# B&R Automation Studio project TD52 (part 57)

#### HiContr.h
```c
/********************************************************************
 * COPYRIGHT -- Bernecker + Rainer Industrie-Elektronik Ges.m.b.H.
 ********************************************************************
 * Program: HiContr
 * File: HiContr.h
 * Author: 106001702
 * Created: Wed Nov 09 12:46:00 2011
 ********************************************************************
 * Header for program HiContr
 ********************************************************************
 * Generated with B&R Automation Studio Target for Simulink V4.2
 * (ERT based)
 ********************************************************************/

#ifndef RTW_HEADER_HiContr_h_
#define RTW_HEADER_HiContr_h_
#ifndef HiContr_COMMON_INCLUDES_
# define HiContr_COMMON_INCLUDES_
#include <math.h>
#include "rtwtypes.h"
#endif                                 /* HiContr_COMMON_INCLUDES_ */

#include "HiContr_types.h"
#include "lHiContr.h"

/* Macros for accessing real-time model data structure */
#ifndef rtmGetErrorStatus
# define rtmGetErrorStatus(rtm)        ((void*) 0)
#endif

#ifndef rtmSetErrorStatus
# define rtmSetErrorStatus(rtm, val)   ((void) 0)
#endif

#ifndef rtmGetStopRequested
# define rtmGetStopRequested(rtm)      ((void*) 0)
#endif

#ifndef MIN
#define MIN(a,b)                       ((a) < (b) ? (a) : (b))
#endif

#ifndef MAX
#define MAX(a,b)                       ((a) > (b) ? (a) : (b))
#endif

/* Block signals (auto storage) */

/* Block states (auto storage) for system '<Root>' */

/* Block signals (auto storage) */
extern BlockIO_HiContr HiContr_B;

/* Block states (auto storage) */
extern D_Work_HiContr HiContr_DWork;

/* Model entry point functions */
extern void HiContr_initialize(struct HiContr* inst);
extern void HiContr_step(struct HiContr* inst);
extern void HiContr_terminate(struct HiContr* inst);

/*-
 * The generated code includes comments that allow you to trace directly
 * back to the appropriate location in the model.  The basic format
 * is <system>/block_name, where system is the system number (uniquely
 * assigned by Simulink) and block_name is the name of the block.
 *
 * Use the MATLAB hilite_system command to trace the generated code back
 * to the model.  For example,
 *
 * hilite_system('<S3>')    - opens system 3
 * hilite_system('<S3>/Kp') - opens and selects block Kp which resides in S3
 *
 * Here is the system hierarchy for this model
 *
 * '<Root>' : 'HiContr'
 * '<S1>'   : 'HiContr/Cyl'
 * '<S2>'   : 'HiContr/Model Info'
 * '<S3>'   : 'HiContr/Cyl/DocBlock'
 * '<S4>'   : 'HiContr/Cyl/GICounter1'
 * '<S5>'   : 'HiContr/Cyl/GlowIgn Integrator'
 * '<S6>'   : 'HiContr/Cyl/Misifire Integrator1'
 * '<S7>'   : 'HiContr/Cyl/Model Info'
 * '<S8>'   : 'HiContr/Cyl/MovingAverage and StdDev'
 * '<S9>'   : 'HiContr/Cyl/Saturation Dynamic1'
 * '<S10>'  : 'HiContr/Cyl/Saturation Dynamic2'
 * '<S11>'  : 'HiContr/Cyl/Saturation Dynamic3'
 * '<S12>'  : 'HiContr/Cyl/Saturation Dynamic4'
 * '<S13>'  : 'HiContr/Cyl/Saturation Dynamic5'
 * '<S14>'  : 'HiContr/Cyl/Threshold'
 * '<S15>'  : 'HiContr/Cyl/Threshold2'
 * '<S16>'  : 'HiContr/Cyl/Threshold3'
 * '<S17>'  : 'HiContr/Cyl/Threshold4'
 * '<S18>'  : 'HiContr/Cyl/Threshold5'
 * '<S19>'  : 'HiContr/Cyl/Threshold6'
 * '<S20>'  : 'HiContr/Cyl/Threshold7'
 * '<S21>'  : 'HiContr/Cyl/Weak Combustion Integrator'
 */
#endif                                 /* RTW_HEADER_HiContr_h_ */
```

#### HiContr_private.h
```c
/********************************************************************
 * COPYRIGHT -- Bernecker + Rainer Industrie-Elektronik Ges.m.b.H.
 ********************************************************************
 * Program: HiContr
 * File: HiContr_private.h
 * Author: 106001702
 * Created: Wed Nov 09 12:46:00 2011
 ********************************************************************
 * Header for program HiContr
 ********************************************************************
 * Generated with B&R Automation Studio Target for Simulink V4.2
 * (ERT based)
 ********************************************************************/

#ifndef RTW_HEADER_HiContr_private_h_
#define RTW_HEADER_HiContr_private_h_
#include "rtwtypes.h"
#include <bur/plctypes.h>
#ifndef __RTWTYPES_H__
#error This file requires rtwtypes.h to be included
#else
#ifdef TMWTYPES_PREVIOUSLY_INCLUDED
#error This file requires rtwtypes.h to be included before tmwtypes.h
#else

/* Check for inclusion of an incorrect version of rtwtypes.h */
#ifndef RTWTYPES_ID_C08S16I32L32N32F1
#error This code was generated with a different "rtwtypes.h" than the file included
#endif                                 /* RTWTYPES_ID_C08S16I32L32N32F1 */
#endif                                 /* TMWTYPES_PREVIOUSLY_INCLUDED */
#endif                                 /* __RTWTYPES_H__ */

#ifndef MIN
#define MIN(a,b)                       ((a) < (b) ? (a) : (b))
#endif

#ifndef MAX
#define MAX(a,b)                       ((a) > (b) ? (a) : (b))
#endif

/* Imported (extern) block parameters */
extern real32_T GIGain;                /* Variable: GIGain
                                        * Referenced by: '<S1>/GIGain (%*100cycles//events)'
                                        */
extern real32_T GIPowGain;             /* Variable: GIPowGain
                                        * Referenced by: '<S1>/GIPowGain (%Pnom*100cycles//events)'
                                        */
extern real32_T MFGain;                /* Variable: MFGain
                                        * Referenced by: '<S1>/MFGain (%*100cycles//events)'
                                        */
extern real32_T MFGainSkipTdown;       /* Variable: MFGainSkipTdown
                                        * Referenced by: '<S1>/MF_Gain_Skip_Tdown'
                                        */
extern real32_T MFThSkipOff;           /* Variable: MFThSkipOff
                                        * Referenced by: '<S1>/Relay1'
                                        */
extern real32_T MFThSkipOn;            /* Variable: MFThSkipOn
                                        * Referenced by: '<S1>/Relay1'
                                        */
extern real32_T PmaxLimReaHys;         /* Variable: PmaxLimReaHys
                                        * Referenced by: '<S1>/Relay'
                                        */
extern real32_T WCGain;                /* Variable: WCGain
                                        * Referenced by: '<S1>/WCGain (bar*100cycles//events)'
                                        */
extern real32_T WCScaling;             /* Variable: WCScaling
                                        * Referenced by: '<S1>/scaling relative to  Pmax at full load (%//bar)'
                                        */

#endif                                 /* RTW_HEADER_HiContr_private_h_ */
```

#### HiContr_types.h
```c
/********************************************************************
 * COPYRIGHT -- Bernecker + Rainer Industrie-Elektronik Ges.m.b.H.
 ********************************************************************
 * Program: HiContr
 * File: HiContr_types.h
 * Author: 106001702
 * Created: Wed Nov 09 12:46:00 2011
 ********************************************************************
 * Header for program HiContr
 ********************************************************************
 * Generated with B&R Automation Studio Target for Simulink V4.2
 * (ERT based)
 ********************************************************************/

#ifndef RTW_HEADER_HiContr_types_h_
#define RTW_HEADER_HiContr_types_h_
#ifndef MIN
#define MIN(a,b)                       ((a) < (b) ? (a) : (b))
#endif

#ifndef MAX
#define MAX(a,b)                       ((a) > (b) ? (a) : (b))
#endif
#endif                                 /* RTW_HEADER_HiContr_types_h_ */
```

#### rtwtypes.h
```c
/********************************************************************
 * COPYRIGHT -- Bernecker + Rainer Industrie-Elektronik Ges.m.b.H.
 ********************************************************************
 * Program: HiContr
 * File: rtwtypes.h
 * Author: 106001702
 * Created: Wed Nov 09 12:46:00 2011
 ********************************************************************
 * Header for program HiContr
 ********************************************************************
 * Generated with B&R Automation Studio Target for Simulink V4.2
 * (ERT based)
 ********************************************************************/

#ifndef __RTWTYPES_H__
#define __RTWTYPES_H__
#ifndef TRUE
# define TRUE                          (1U)
#endif

#ifndef FALSE
# define FALSE                         (0U)
#endif

#ifndef __TMWTYPES__
#define __TMWTYPES__
#include <limits.h>

/*=======================================================================*
 * Target hardware information
 *   Device type: Intel->x86/Pentium
 *   Number of bits:     char:   8    short:   16    int:  32
 *                       long:  32
 *                       native word size:  32
 *   Byte ordering: LittleEndian
 *   Signed integer division rounds to: Zero
 *   Shift right on a signed integer as arithmetic shift: on
 *=======================================================================*/

/*=======================================================================*
 * Fixed width word size data types:                                     *
 *   int8_T, int16_T, int32_T     - signed 8, 16, or 32 bit integers     *
 *   uint8_T, uint16_T, uint32_T  - unsigned 8, 16, or 32 bit integers   *
 *   real32_T, real64_T           - 32 and 64 bit floating point numbers *
 *=======================================================================*/
typedef signed char int8_T;
typedef unsigned char uint8_T;
typedef short int16_T;
typedef unsigned short uint16_T;
typedef int int32_T;
typedef unsigned int uint32_T;
typedef float real32_T;
typedef double real64_T;

/*===========================================================================*
 * Generic type definitions: real_T, time_T, boolean_T, int_T, uint_T,       *
 *                           ulong_T, char_T and byte_T.                     *
 *===========================================================================*/
typedef double real_T;
typedef double time_T;
typedef unsigned char boolean_T;
typedef int int_T;
typedef unsigned int uint_T;
typedef unsigned long ulong_T;
typedef char char_T;
typedef unsigned char uchar_T;
typedef char_T byte_T;

/*=======================================================================*
 * Min and Max:                                                          *
 *   int8_T, int16_T, int32_T     - signed 8, 16, or 32 bit integers     *
 *   uint8_T, uint16_T, uint32_T  - unsigned 8, 16, or 32 bit integers   *
 *=======================================================================*/
#define MAX_int8_T                     ((int8_T)(127))
#define MIN_int8_T                     ((int8_T)(-128))
#define MAX_uint8_T                    ((uint8_T)(255U))
#define MIN_uint8_T                    ((uint8_T)(0U))
#define MAX_int16_T                    ((int16_T)(32767))
#define MIN_int16_T                    ((int16_T)(-32768))
#define MAX_uint16_T                   ((uint16_T)(65535U))
#define MIN_uint16_T                   ((uint16_T)(0U))
#define MAX_int32_T                    ((int32_T)(2147483647))
#define MIN_int32_T                    ((int32_T)(-2147483647-1))
#define MAX_uint32_T                   ((uint32_T)(0xFFFFFFFFU))
#define MIN_uint32_T                   ((uint32_T)(0U))

/* Logical type definitions */
#if (!defined(__cplusplus)) && (!defined(__true_false_are_keywords))
#  ifndef false
#   define false                       (0U)
#  endif

#  ifndef true
#   define true                        (1U)
#  endif
#endif

/*
 * Simulink Coder assumes the code is compiled on a target using a 2's complement representation
 * for signed integer values.
 */
#if ((SCHAR_MIN + 1) != -SCHAR_MAX)
#error "This code must be compiled using a 2's complement representation for signed integer values"
#endif

/* This ID is used to detect inclusion of an incompatible rtwtypes.h */
#define RTWTYPES_ID_C08S16I32L32N32F1
#else                                  /* __TMWTYPES__ */
#define TMWTYPES_PREVIOUSLY_INCLUDED
#endif                                 /* __TMWTYPES__ */

/* Block D-Work pointer type */
typedef void * pointer_T;

/* Simulink specific types */
#ifndef __SIMSTRUC_TYPES_H__
#define __SIMSTRUC_TYPES_H__

/* Trigger directions: falling, either, and rising */
typedef enum {
  FALLING_ZERO_CROSSING = -1,
  ANY_ZERO_CROSSING = 0,
  RISING_ZERO_CROSSING = 1
} ZCDirection;

/* Previous state of a trigger signal */
typedef uint8_T ZCSigState;

/* Initial value of a trigger zero crossing signal */
#define UNINITIALIZED_ZCSIG            0x03U
#define NEG_ZCSIG                      0x02U
#define POS_ZCSIG                      0x01U
#define ZERO_ZCSIG                     0x00U

/* Current state of a trigger signal */
typedef enum {
  FALLING_ZCEVENT = -1,
  NO_ZCEVENT = 0,
  RISING_ZCEVENT = 1
} ZCEventType;

#endif                                 /* __SIMSTRUC_TYPES_H__ */
#endif                                 /* __RTWTYPES_H__ */

#ifndef MIN
#define MIN(a,b)                       ((a) < (b) ? (a) : (b))
#endif

#ifndef MAX
#define MAX(a,b)                       ((a) > (b) ? (a) : (b))
#endif
```

#### HiContr.c
```c
/********************************************************************
 * COPYRIGHT -- Bernecker + Rainer Industrie-Elektronik Ges.m.b.H.
 ********************************************************************
 * Program: HiContr
 * File: HiContr.c
 * Author: 106001702
 * Created: Wed Nov 09 12:46:00 2011
 ********************************************************************
 * Implementation of program HiContr
 ********************************************************************
 * Generated with B&R Automation Studio Target for Simulink V4.2
 * (ERT based)
 ********************************************************************/
#include "HiContr.h"
#include "HiContr_private.h"

/*  Defines */

/*  Data Types */

/**************************** GLOBAL DATA *************************************/
/*  Definitions */

/* Block signals (auto storage) */

/* Block states (auto storage) */

/*  Declarations  */

/***************************** FILE SCOPE DATA ********************************/

/*************************** FUNCTIONS ****************************************/

/* Model step function */
void HiContr_step(struct HiContr* inst)
{
  /* local block i/o variables */
  boolean_T rtb_Compare_j;
  real32_T rtb_Switch1;
  boolean_T rtb_Compare;
  boolean_T rtb_LogicalOperator6;
  real32_T rtb_invert;
  boolean_T rtb_LogicalOperator3;
  real_T rtb_Divide3_g;
  real32_T rtb_MathFunction[100];
  real32_T rtb_Sum;
  real32_T rtb_Divide2;
  real32_T rtb_Add7;
  boolean_T rtb_LogicalOperator1;
  boolean_T rtb_LogicalOperator11;
  boolean_T rtb_LogicalOperator;
  boolean_T rtb_BitwiseOperator2;
  boolean_T rtb_BitwiseOperator1;
  real32_T rtb_Add8;
  real_T rtb_Divide3_d;
  real_T rtb_Divide3_p;
  real_T rtb_Add;
  int32_T i;
  int16_T tmp;

  /* S-Function (bur_in): '<S1>/Input17' */
  inst->bur_HiContr_B.Input17 = inst->GIThPIDUR;

  /* S-Function (bur_in): '<Root>/Input5' */
  inst->bur_HiContr_B.Input5_c = inst->EngStopErrAck;

  /* DiscreteIntegrator: '<S5>/Discrete-Time Integrator' */
  if (inst->bur_HiContr_B.Input5_c || (inst->bur_HiContr_DWork.DiscreteTimeIntegrator_PrevRese != 0))
  {
    inst->bur_HiContr_DWork.DiscreteTimeIntegrator_DSTATE = 0.0F;
  }

  if (inst->bur_HiContr_DWork.DiscreteTimeIntegrator_DSTATE >= 100.0F) {
    inst->bur_HiContr_DWork.DiscreteTimeIntegrator_DSTATE = 100.0F;
  } else {
    if (inst->bur_HiContr_DWork.DiscreteTimeIntegrator_DSTATE <= 0.0F) {
      inst->bur_HiContr_DWork.DiscreteTimeIntegrator_DSTATE = 0.0F;
    }
  }

  inst->bur_HiContr_B.DiscreteTimeIntegrator = inst->bur_HiContr_DWork.DiscreteTimeIntegrator_DSTATE;

  /* End of DiscreteIntegrator: '<S5>/Discrete-Time Integrator' */

  /* Sum: '<S1>/Add5' */
  rtb_Switch1 = inst->bur_HiContr_B.DiscreteTimeIntegrator - inst->bur_HiContr_B.Input17;

  /* S-Function (bur_in): '<Root>/Input9' */
  inst->bur_HiContr_B.Input9_a = inst->GIContrEnable;

  /* Logic: '<S1>/Logical Operator6' incorporates:
   *  Constant: '<S16>/Constant'
   *  RelationalOperator: '<S16>/Compare'
   */
  rtb_LogicalOperator6 = ((rtb_Switch1 > 0.0F) && inst->bur_HiContr_B.Input9_a);

  /* Switch: '<S1>/Switch2' incorporates:
   *  Constant: '<S1>/Constant2'
   */
  if (!rtb_LogicalOperator6) {
    rtb_Switch1 = 0.0F;
  }

  /* End of Switch: '<S1>/Switch2' */

  /* Gain: '<S1>/invert' incorporates:
   *  Gain: '<S1>/GIGain (%*100cycles//events)'
   */
  rtb_invert = -(inst->GIGain * rtb_Switch1);

  /* S-Function (bur_in): '<S1>/Input13' */
  inst->bur_HiContr_B.Input13 = inst->GIPIDURLimMin;

  /* Switch: '<S12>/Switch2' incorporates:
   *  Constant: '<S1>/Constant6'
   *  RelationalOperator: '<S12>/LowerRelop1'
   *  RelationalOperator: '<S12>/UpperRelop'
   *  Switch: '<S12>/Switch'
   */
  if (rtb_invert > 0.0F) {
    inst->bur_HiContr_B.Switch2 = 0.0F;
  } else if (rtb_invert < inst->bur_HiContr_B.Input13) {
    /* Switch: '<S12>/Switch' */
    inst->bur_HiContr_B.Switch2 = inst->bur_HiContr_B.Input13;
  } else {
    inst->bur_HiContr_B.Switch2 = rtb_invert;
  }

  /* End of Switch: '<S12>/Switch2' */

  /* S-Function (bur_out): '<S1>/Output1' */
  inst->PIDUROffsetGI = inst->bur_HiContr_B.Switch2;

  /* S-Function (bur_in): '<S1>/Input11' */
  inst->bur_HiContr_B.Input11 = inst->MFPIDURLimMax;

  /* S-Function (bur_in): '<S1>/Input14' */
  inst->bur_HiContr_B.Input14 = inst->MFThPIDUR;

  /* DiscreteIntegrator: '<S6>/Discrete-Time Integrator' */
  if (inst->bur_HiContr_B.Input5_c || (inst->bur_HiContr_DWork.DiscreteTimeIntegrator_PrevRe_f != 0))
  {
    inst->bur_HiContr_DWork.DiscreteTimeIntegrator_DSTATE_e = 0.0F;
  }

  if (inst->bur_HiContr_DWork.DiscreteTimeIntegrator_DSTATE_e >= 100.0F) {
    inst->bur_HiContr_DWork.DiscreteTimeIntegrator_DSTATE_e = 100.0F;
  } else {
    if (inst->bur_HiContr_DWork.DiscreteTimeIntegrator_DSTATE_e <= 0.0F) {
      inst->bur_HiContr_DWork.DiscreteTimeIntegrator_DSTATE_e = 0.0F;
    }
  }

  inst->bur_HiContr_B.DiscreteTimeIntegrator_d =
    inst->bur_HiContr_DWork.DiscreteTimeIntegrator_DSTATE_e;

  /* End of DiscreteIntegrator: '<S6>/Discrete-Time Integrator' */

  /* Sum: '<S1>/Add2' */
  rtb_Switch1 = inst->bur_HiContr_B.DiscreteTimeIntegrator_d - inst->bur_HiContr_B.Input14;

  /* S-Function (bur_in): '<Root>/Input7' */
  inst->bur_HiContr_B.Input7_c = inst->MFContrEnable;

  /* Logic: '<S1>/Logical Operator3' incorporates:
   *  Constant: '<S14>/Constant'
   *  RelationalOperator: '<S14>/Compare'
   */
  rtb_LogicalOperator3 = ((rtb_Switch1 > 0.0F) && inst->bur_HiContr_B.Input7_c);

  /* Switch: '<S1>/Switch' incorporates:
   *  Constant: '<S1>/Constant'
   */
  if (!rtb_LogicalOperator3) {
    rtb_Switch1 = 0.0F;
  }

  /* End of Switch: '<S1>/Switch' */

  /* Gain: '<S1>/MFGain (%*100cycles//events)' */
  rtb_invert = inst->MFGain * rtb_Switch1;

  /* Switch: '<S9>/Switch2' incorporates:
   *  Constant: '<S1>/Constant7'
   *  RelationalOperator: '<S9>/LowerRelop1'
   *  RelationalOperator: '<S9>/UpperRelop'
   *  Switch: '<S9>/Switch'
   */
  if (rtb_invert > inst->bur_HiContr_B.Input11) {
    inst->bur_HiContr_B.Switch2_e = inst->bur_HiContr_B.Input11;
  } else if (rtb_invert < 0.0F) {
    /* Switch: '<S9>/Switch' incorporates:
     *  Constant: '<S1>/Constant7'
     */
    inst->bur_HiContr_B.Switch2_e = 0.0F;
  } else {
    inst->bur_HiContr_B.Switch2_e = rtb_invert;
  }

  /* End of Switch: '<S9>/Switch2' */

  /* S-Function (bur_out): '<S1>/Output2' */
  inst->PIDUROffsetMF = inst->bur_HiContr_B.Switch2_e;

  /* S-Function (bur_out): '<S1>/Output3' */
  inst->MFIntOut = inst->bur_HiContr_B.DiscreteTimeIntegrator_d;

  /* DiscreteIntegrator: '<S21>/Discrete-Time Integrator' */
  if (inst->bur_HiContr_B.Input5_c || (inst->bur_HiContr_DWork.DiscreteTimeIntegrator_PrevRe_c != 0))
  {
    inst->bur_HiContr_DWork.DiscreteTimeIntegrator_DSTATE_c = 0.0F;
  }

  if (inst->bur_HiContr_DWork.DiscreteTimeIntegrator_DSTATE_c >= 100.0F) {
    inst->bur_HiContr_DWork.DiscreteTimeIntegrator_DSTATE_c = 100.0F;
  } else {
    if (inst->bur_HiContr_DWork.DiscreteTimeIntegrator_DSTATE_c <= 0.0F) {
      inst->bur_HiContr_DWork.DiscreteTimeIntegrator_DSTATE_c = 0.0F;
    }
  }

  inst->bur_HiContr_B.DiscreteTimeIntegrator_l =
    inst->bur_HiContr_DWork.DiscreteTimeIntegrator_DSTATE_c;

  /* End of DiscreteIntegrator: '<S21>/Discrete-Time Integrator' */

  /* S-Function (bur_out): '<S1>/Output4' */
  inst->WCIntOut = inst->bur_HiContr_B.DiscreteTimeIntegrator_l;

  /* S-Function (bur_out): '<S1>/Output5' */
  inst->GIIntOut = inst->bur_HiContr_B.DiscreteTimeIntegrator;

  /* S-Function (bur_in): '<Root>/Input10' */
  inst->bur_HiContr_B.Input10_h = inst->PmaxLimContrEnable;

  /* S-Function (bur_in): '<Root>/Input11' */
  inst->bur_HiContr_B.Input11_h = inst->PmaxLimDiane;

  /* S-Function (bur_in): '<S1>/Input7' */
  inst->bur_HiContr_B.Input7 = inst->PmaxSDLimMar;

  /* Sum: '<S1>/Subtract' */
  rtb_invert = inst->bur_HiContr_B.Input11_h - inst->bur_HiContr_B.Input7;

  /* Sum: '<S8>/Sum of Elements' incorporates:
   *  S-Function (sfix_udelay): '<S8>/Tapped Delay set as N_cyc!!!'
   */
  rtb_Divide3_g = inst->bur_HiContr_DWork.TappedDelaysetasN_cyc_X[0];
  for (i = 0; i < 99; i++) {
    rtb_Divide3_g += (real_T)inst->bur_HiContr_DWork.TappedDelaysetasN_cyc_X[i + 1];
  }

  /* End of Sum: '<S8>/Sum of Elements' */

  /* Product: '<S8>/Divide' incorporates:
   *  Constant: '<S8>/set as Ncyc!!!'
   */
  inst->bur_HiContr_B.Divide = (real32_T)(rtb_Divide3_g / 100.0);

  /* Math: '<S8>/Math Function'
   *
   * About '<S8>/Math Function':
   *  Operator: magnitude^2
   */
  for (i = 0; i < 100; i++) {
    /* Sum: '<S8>/Add' incorporates:
     *  S-Function (sfix_udelay): '<S8>/Tapped Delay set as N_cyc!!!'
     */
    rtb_Switch1 = inst->bur_HiContr_DWork.TappedDelaysetasN_cyc_X[i] - inst->bur_HiContr_B.Divide;
    rtb_MathFunction[i] = rtb_Switch1 * rtb_Switch1;
  }

  /* End of Math: '<S8>/Math Function' */

  /* Sum: '<S8>/Sum of Elements2' */
  rtb_Switch1 = rtb_MathFunction[0];
  for (i = 0; i < 99; i++) {
    rtb_Switch1 += rtb_MathFunction[i + 1];
  }

  /* End of Sum: '<S8>/Sum of Elements2' */

  /* Sqrt: '<S8>/Sqrt' incorporates:
   *  Constant: '<S8>/set as Ncyc!!!'
   *  Product: '<S8>/Divide1'
   */
  inst->bur_HiContr_B.Sqrt = (real32_T)sqrt((real32_T)((real_T)rtb_Switch1 / 100.0));

  /* S-Function (bur_in): '<S1>/Input8' */
  inst->bur_HiContr_B.Input8 = inst->PmaxStdevFact;

  /* Sum: '<S1>/Sum' incorporates:
   *  Product: '<S1>/Product2'
   *  Sum: '<S1>/Add'
   */
  rtb_Sum = rtb_invert - (inst->bur_HiContr_B.Sqrt * inst->bur_HiContr_B.Input8 + inst->bur_HiContr_B.Divide);

  /* S-Function (bur_in): '<S1>/Input9' */
  inst->bur_HiContr_B.Input9 = inst->PmaxContrGain;

  /* Product: '<S1>/Product1' incorporates:
   *  Product: '<S1>/Product3'
   */
  rtb_invert = inst->bur_HiContr_B.Input10_h ? rtb_Sum * inst->bur_HiContr_B.Input9 : 0.0F;

  /* S-Function (bur_in): '<S1>/Input10' */
  inst->bur_HiContr_B.Input10 = inst->PmaxContrLimMin;

  /* Switch: '<S10>/Switch2' incorporates:
   *  Constant: '<S1>/Constant4'
   *  RelationalOperator: '<S10>/LowerRelop1'
   *  RelationalOperator: '<S10>/UpperRelop'
   *  Switch: '<S10>/Switch'
   */
  if (rtb_invert > 0.0F) {
    inst->bur_HiContr_B.Switch2_k = 0.0F;
  } else if (rtb_invert < inst->bur_HiContr_B.Input10) {
    /* Switch: '<S10>/Switch' */
    inst->bur_HiContr_B.Switch2_k = inst->bur_HiContr_B.Input10;
  } else {
    inst->bur_HiContr_B.Switch2_k = rtb_invert;
  }

  /* End of Switch: '<S10>/Switch2' */

  /* S-Function (bur_out): '<S1>/Output6' */
  inst->PIDUROffsetPmax = inst->bur_HiContr_B.Switch2_k;

  /* S-Function (bur_in): '<S1>/Input19' */
  inst->bur_HiContr_B.Input19 = inst->GIThSkipReset;

  /* RelationalOperator: '<S18>/Compare' incorporates:
   *  Constant: '<S18>/Constant'
   *  Sum: '<S1>/Add1'
   */
  rtb_Compare_j = (inst->bur_HiContr_B.DiscreteTimeIntegrator - inst->bur_HiContr_B.Input19 < 0.0F);

  /* DiscreteIntegrator: '<S4>/Discrete-Time Integrator' */
  if (rtb_Compare_j || (inst->bur_HiContr_DWork.DiscreteTimeIntegrator_PrevRe_n != 0)) {
    inst->bur_HiContr_DWork.DiscreteTimeIntegrator_DSTATE_n = 0.0F;
  }

  if (inst->bur_HiContr_DWork.DiscreteTimeIntegrator_DSTATE_n >= 100.0F) {
    inst->bur_HiContr_DWork.DiscreteTimeIntegrator_DSTATE_n = 100.0F;
  } else {
    if (inst->bur_HiContr_DWork.DiscreteTimeIntegrator_DSTATE_n <= 0.0F) {
      inst->bur_HiContr_DWork.DiscreteTimeIntegrator_DSTATE_n = 0.0F;
    }
  }

  inst->bur_HiContr_B.DiscreteTimeIntegrator_dl =
    inst->bur_HiContr_DWork.DiscreteTimeIntegrator_DSTATE_n;

  /* End of DiscreteIntegrator: '<S4>/Discrete-Time Integrator' */

  /* S-Function (bur_out): '<S1>/Output7' */
  inst->GICountOut = inst->bur_HiContr_B.DiscreteTimeIntegrator_dl;

  /* S-Function (bur_out): '<S1>/Output8' */
  inst->PmaxAv = inst->bur_HiContr_B.Divide;

  /* S-Function (bur_out): '<S1>/Output9' */
  inst->PmaxStd = inst->bur_HiContr_B.Sqrt;

  /* S-Function (bur_in): '<S1>/Input16' */
  inst->bur_HiContr_B.Input16 = inst->WCThPmax;

  /* Sum: '<S1>/Add4' */
  rtb_Switch1 = inst->bur_HiContr_B.DiscreteTimeIntegrator_l - inst->bur_HiContr_B.Input16;

  /* S-Function (bur_in): '<S1>/Input18' */
  inst->bur_HiContr_B.Input18 = inst->GIThSkip;

  /* Sum: '<S1>/Add6' */
  rtb_invert = inst->bur_HiContr_B.DiscreteTimeIntegrator - inst->bur_HiContr_B.Input18;

  /* S-Function (bur_in): '<S1>/Input21' */
  inst->bur_HiContr_B.Input21 = inst->GIThCount;

  /* Sum: '<S1>/Add7' */
  rtb_Add7 = inst->bur_HiContr_B.DiscreteTimeIntegrator_dl - inst->bur_HiContr_B.Input21;

  /* Relay: '<S1>/Relay1' */
  if (inst->bur_HiContr_B.DiscreteTimeIntegrator_d >= inst->MFThSkipOn) {
    inst->bur_HiContr_DWork.Relay1_Mode = TRUE;
  } else {
    if (inst->bur_HiContr_B.DiscreteTimeIntegrator_d <= inst->MFThSkipOff) {
      inst->bur_HiContr_DWork.Relay1_Mode = FALSE;
    }
  }

  if (inst->bur_HiContr_DWork.Relay1_Mode) {
    rtb_Divide2 = 1.0F;
  } else {
    rtb_Divide2 = 0.0F;
  }

  /* End of Relay: '<S1>/Relay1' */

  /* Sum: '<S1>/Add8' incorporates:
   *  Constant: '<S1>/Constant3'
   *  Gain: '<S1>/MF_Gain_Skip_Tdown'
   */
  rtb_Add8 = inst->MFGainSkipTdown * rtb_Divide2 + 1.0F;

  /* S-Function (bur_in): '<Root>/Input1' */
  inst->bur_HiContr_B.Input1_h = inst->Misfire2;

  /* S-Function (sfix_bitop): '<S1>/Bitwise Operator' */
  rtb_Compare = !inst->bur_HiContr_B.Input1_h;

  /* S-Function (bur_in): '<Root>/Input20' */
  inst->bur_HiContr_B.Input20_o = inst->Misfire1;

  /* S-Function (sfix_bitop): '<S1>/Bitwise Operator1' */
  rtb_BitwiseOperator1 = !inst->bur_HiContr_B.Input20_o;

  /* RelationalOperator: '<S19>/Compare' incorporates:
   *  Constant: '<S19>/Constant'
   */
  rtb_LogicalOperator1 = (rtb_Add7 > 0.0F);

  /* S-Function (sfix_bitop): '<S1>/Bitwise Operator2' */
  rtb_BitwiseOperator2 = !rtb_LogicalOperator1;

  /* S-Function (bur_in): '<Root>/Input4' */
  inst->bur_HiContr_B.Input4_d = inst->SensSignFault;

  /* S-Function (sfix_bitop): '<S1>/Bitwise Operator3' */
  rtb_LogicalOperator = !inst->bur_HiContr_B.Input4_d;

  /* S-Function (bur_in): '<S1>/Input6' */
  inst->bur_HiContr_B.Input6 = inst->TGICount;

  /* Logic: '<S1>/Logical Operator9' incorporates:
   *  Constant: '<S17>/Constant'
   *  RelationalOperator: '<S17>/Compare'
   */
  rtb_LogicalOperator11 = (inst->bur_HiContr_B.Input9_a && (rtb_invert > 0.0F));

  /* Sum: '<S4>/Add' incorporates:
   *  Constant: '<S1>/Constant9'
   *  Product: '<S4>/Divide'
   *  Product: '<S4>/Divide2'
   */
  rtb_Add = rtb_LogicalOperator11 ? 1.0 / (real_T)inst->bur_HiContr_B.Input6 : 0.0;

  /* Switch: '<S1>/Switch3' incorporates:
   *  Constant: '<S1>/Constant12'
   *  Logic: '<S1>/Logical Operator10'
   */
  if (rtb_LogicalOperator1 && inst->bur_HiContr_B.Input9_a) {
    /* Switch: '<S13>/Switch2' incorporates:
     *  Constant: '<S1>/Constant10'
     *  Constant: '<S1>/Constant11'
     *  RelationalOperator: '<S13>/LowerRelop1'
     *  RelationalOperator: '<S13>/UpperRelop'
     *  Switch: '<S13>/Switch'
     */
    if (rtb_invert > 100.0F) {
      rtb_invert = 100.0F;
    } else {
      if (rtb_invert < 0.0F) {
        /* Switch: '<S13>/Switch' incorporates:
         *  Constant: '<S1>/Constant10'
         */
        rtb_invert = 0.0F;
      }
    }

    /* End of Switch: '<S13>/Switch2' */
  } else {
    rtb_invert = 0.0F;
  }

  /* End of Switch: '<S1>/Switch3' */

  /* Gain: '<S1>/GIPowGain (%Pnom*100cycles//events)' */
  inst->bur_HiContr_B.GIPowGainPnom100cyclesevents = inst->GIPowGain * rtb_invert;

  /* S-Function (bur_in): '<S1>/Input5' */
  inst->bur_HiContr_B.Input5 = inst->TdownGI;

  /* Product: '<S5>/Divide1' incorporates:
   *  Constant: '<S5>/Constant'
   */
  rtb_Divide3_g = 1.0 / (real_T)inst->bur_HiContr_B.Input5;

  /* S-Function (bur_in): '<Root>/Input2' */
  inst->bur_HiContr_B.Input2_g = inst->GlowIgn;

  /* S-Function (bur_in): '<S1>/Input4' */
  inst->bur_HiContr_B.Input4 = inst->TupGI;

  /* Sum: '<S5>/Add' incorporates:
   *  Product: '<S5>/Divide'
   *  Product: '<S5>/Divide2'
   *  Product: '<S5>/Divide3'
   */
  rtb_Divide3_g = (real_T)(rtb_LogicalOperator ? (real32_T)inst->bur_HiContr_B.Input2_g /
    inst->bur_HiContr_B.Input4 : 0.0F) - (rtb_LogicalOperator ? rtb_Divide3_g : 0.0);

  /* S-Function (bur_in): '<S1>/Input1' */
  inst->bur_HiContr_B.Input1 = inst->TdownMF;

  /* S-Function (bur_in): '<S1>/Input12' */
  inst->bur_HiContr_B.Input12 = inst->WCPmaxLimMax;

  /* S-Function (bur_in): '<S1>/Input2' */
  inst->bur_HiContr_B.Input2 = inst->TupWC;

  /* S-Function (bur_in): '<S1>/Input20' */
  inst->bur_HiContr_B.Input20 = inst->TupMF;

  /* S-Function (bur_in): '<S1>/Input3' */
  inst->bur_HiContr_B.Input3 = inst->TdownWC;

  /* Logic: '<S1>/Logical Operator' */
  rtb_LogicalOperator = (inst->bur_HiContr_B.Input20_o && inst->bur_HiContr_B.Input1_h);

  /* Logic: '<S1>/Logical Operator1' */
  rtb_LogicalOperator1 = (inst->bur_HiContr_B.Input20_o && rtb_Compare);

  /* S-Function (bur_in): '<Root>/Input6' */
  inst->bur_HiContr_B.Input6_a = inst->KnockCountMeasAct;

  /* Relay: '<S1>/Relay' */
  if (rtb_Sum >= inst->PmaxLimReaHys) {
    inst->bur_HiContr_DWork.Relay_Mode = TRUE;
  } else {
    if (rtb_Sum <= 0.0F) {
      inst->bur_HiContr_DWork.Relay_Mode = FALSE;
    }
  }

  if (inst->bur_HiContr_DWork.Relay_Mode) {
    tmp = 0;
  } else {
    tmp = 1;
  }

  /* End of Relay: '<S1>/Relay' */

  /* RelationalOperator: '<S20>/Compare' incorporates:
   *  Constant: '<S20>/Constant'
   */
  inst->bur_HiContr_B.Compare = (tmp > 0);

  /* Logic: '<S1>/Logical Operator13' incorporates:
   *  Logic: '<S1>/Logical Operator14'
   *  Logic: '<S1>/Logical Operator5'
   */
  inst->bur_HiContr_B.LogicalOperator13 = ((inst->bur_HiContr_B.Input7_c && (rtb_Divide2 != 0.0F)) ||
                                 (rtb_LogicalOperator11 && rtb_BitwiseOperator2));

  /* S-Function (bur_in): '<Root>/Input12' */
  inst->bur_HiContr_B.Input12_e = inst->SkipCylExt;

  /* Logic: '<S1>/Logical Operator11' incorporates:
   *  Logic: '<S1>/Logical Operator12'
   */
  rtb_LogicalOperator11 = !(inst->bur_HiContr_B.Input6_a || rtb_LogicalOperator6 ||
    inst->bur_HiContr_B.Compare || inst->bur_HiContr_B.Input4_d || (inst->bur_HiContr_B.LogicalOperator13 ||
    inst->bur_HiContr_B.Input12_e));

  /* Logic: '<S1>/Logical Operator2' */
  inst->bur_HiContr_B.LogicalOperator2 = (rtb_BitwiseOperator1 && inst->bur_HiContr_B.Input1_h);

  /* S-Function (bur_in): '<Root>/Input8' */
  inst->bur_HiContr_B.Input8_f = inst->WCContrEnable;

  /* Logic: '<S1>/Logical Operator7' */
  inst->bur_HiContr_B.LogicalOperator7 = (rtb_LogicalOperator3 || rtb_LogicalOperator6 ||
    inst->bur_HiContr_B.Compare || inst->bur_HiContr_B.Input4_d);

  /* Logic: '<S1>/Logical Operator8' */
  inst->bur_HiContr_B.LogicalOperator8 = (rtb_LogicalOperator3 || rtb_LogicalOperator6 ||
    inst->bur_HiContr_B.Compare || inst->bur_HiContr_B.Input4_d);

  /* MinMax: '<S1>/MinMax' */
  if (inst->bur_HiContr_B.Switch2_k <= inst->bur_HiContr_B.Switch2) {
    rtb_Add7 = inst->bur_HiContr_B.Switch2_k;
  } else {
    rtb_Add7 = inst->bur_HiContr_B.Switch2;
  }

  /* Product: '<S6>/Divide3' incorporates:
   *  Constant: '<S6>/Constant'
   *  Product: '<S1>/Product'
   *  Product: '<S6>/Divide1'
   */
  rtb_Divide3_d = 1.0 / (real_T)(inst->bur_HiContr_B.Input1 * rtb_Add8);

  /* Product: '<S6>/Divide2' incorporates:
   *  Product: '<S6>/Divide'
   */
  rtb_Divide2 = rtb_LogicalOperator11 ? (real32_T)rtb_LogicalOperator /
    inst->bur_HiContr_B.Input20 : 0.0F;

  /* Switch: '<S1>/Switch1' incorporates:
   *  Constant: '<S15>/Constant'
   *  Constant: '<S1>/Constant1'
   *  Logic: '<S1>/Logical Operator4'
   *  RelationalOperator: '<S15>/Compare'
   */
  if (!((rtb_Switch1 > 0.0F) && inst->bur_HiContr_B.Input8_f)) {
    rtb_Switch1 = 0.0F;
  }

  /* End of Switch: '<S1>/Switch1' */

  /* Gain: '<S1>/scaling relative to  Pmax at full load (%//bar)' incorporates:
   *  Gain: '<S1>/WCGain (bar*100cycles//events)'
   */
  rtb_invert = inst->WCGain * rtb_Switch1 * inst->WCScaling;

  /* Switch: '<S11>/Switch2' incorporates:
   *  Constant: '<S1>/Constant8'
   *  RelationalOperator: '<S11>/LowerRelop1'
   *  RelationalOperator: '<S11>/UpperRelop'
   *  Switch: '<S11>/Switch'
   */
  if (rtb_invert > inst->bur_HiContr_B.Input12) {
    inst->bur_HiContr_B.Switch2_a = inst->bur_HiContr_B.Input12;
  } else if (rtb_invert < 0.0F) {
    /* Switch: '<S11>/Switch' incorporates:
     *  Constant: '<S1>/Constant8'
     */
    inst->bur_HiContr_B.Switch2_a = 0.0F;
  } else {
    inst->bur_HiContr_B.Switch2_a = rtb_invert;
  }

  /* End of Switch: '<S11>/Switch2' */

  /* Switch: '<S1>/Switch4' incorporates:
   *  MinMax: '<S1>/MinMax'
   */
  if (rtb_Add7 >= 0.0F) {
    inst->bur_HiContr_B.Switch4 = inst->bur_HiContr_B.Switch2_e;
  } else {
    inst->bur_HiContr_B.Switch4 = rtb_Add7;
  }

  /* End of Switch: '<S1>/Switch4' */

  /* Product: '<S21>/Divide3' incorporates:
   *  Constant: '<S21>/Constant'
   *  Product: '<S21>/Divide1'
   */
  rtb_Divide3_p = 1.0 / (real_T)inst->bur_HiContr_B.Input3;

  /* Product: '<S21>/Divide2' incorporates:
   *  Product: '<S21>/Divide'
   */
  rtb_invert = rtb_LogicalOperator11 ? (real32_T)rtb_LogicalOperator1 /
    inst->bur_HiContr_B.Input2 : 0.0F;

  /* S-Function (bur_out): '<Root>/Output1' */
  inst->FaultMFSign = inst->bur_HiContr_B.LogicalOperator2;

  /* S-Function (bur_out): '<Root>/Output2' */
  inst->MFB50Freeze = inst->bur_HiContr_B.LogicalOperator7;

  /* S-Function (bur_out): '<Root>/Output3' */
  inst->OptPIDFreeze = inst->bur_HiContr_B.LogicalOperator8;

  /* S-Function (bur_out): '<Root>/Output4' */
  inst->PIDUROffsetCyl = inst->bur_HiContr_B.Switch4;

  /* S-Function (bur_out): '<Root>/Output6' */
  inst->PmaxStabLayOffset = inst->bur_HiContr_B.Switch2_a;

  /* S-Function (bur_out): '<Root>/Output7' */
  inst->PmaxLimReached = inst->bur_HiContr_B.Compare;

  /* S-Function (bur_out): '<Root>/Output8' */
  inst->SkipCyl = inst->bur_HiContr_B.LogicalOperator13;

  /* S-Function (bur_out): '<Root>/Output9' */
  inst->PowRedCyl = inst->bur_HiContr_B.GIPowGainPnom100cyclesevents;

  /* S-Function (bur_in): '<Root>/Input3' */
  inst->bur_HiContr_B.Input3_g = inst->Pmax;

  /* Update for DiscreteIntegrator: '<S5>/Discrete-Time Integrator' */
  if (!inst->bur_HiContr_B.Input5_c) {
    inst->bur_HiContr_DWork.DiscreteTimeIntegrator_DSTATE += (real32_T)(0.01 *
      rtb_Divide3_g);
    if (inst->bur_HiContr_DWork.DiscreteTimeIntegrator_DSTATE >= 100.0F) {
      inst->bur_HiContr_DWork.DiscreteTimeIntegrator_DSTATE = 100.0F;
    } else {
      if (inst->bur_HiContr_DWork.DiscreteTimeIntegrator_DSTATE <= 0.0F) {
        inst->bur_HiContr_DWork.DiscreteTimeIntegrator_DSTATE = 0.0F;
      }
    }
  }

  if (inst->bur_HiContr_B.Input5_c) {
    inst->bur_HiContr_DWork.DiscreteTimeIntegrator_PrevRese = 1;
  } else {
    inst->bur_HiContr_DWork.DiscreteTimeIntegrator_PrevRese = 0;
  }

  /* End of Update for DiscreteIntegrator: '<S5>/Discrete-Time Integrator' */

  /* Update for DiscreteIntegrator: '<S6>/Discrete-Time Integrator' incorporates:
   *  Sum: '<S6>/Add'
   */
  if (!inst->bur_HiContr_B.Input5_c) {
    inst->bur_HiContr_DWork.DiscreteTimeIntegrator_DSTATE_e += (real32_T)(((real_T)
      rtb_Divide2 - rtb_Divide3_d) * 0.01);
    if (inst->bur_HiContr_DWork.DiscreteTimeIntegrator_DSTATE_e >= 100.0F) {
      inst->bur_HiContr_DWork.DiscreteTimeIntegrator_DSTATE_e = 100.0F;
    } else {
      if (inst->bur_HiContr_DWork.DiscreteTimeIntegrator_DSTATE_e <= 0.0F) {
        inst->bur_HiContr_DWork.DiscreteTimeIntegrator_DSTATE_e = 0.0F;
      }
    }
  }

  if (inst->bur_HiContr_B.Input5_c) {
    inst->bur_HiContr_DWork.DiscreteTimeIntegrator_PrevRe_f = 1;
  } else {
    inst->bur_HiContr_DWork.DiscreteTimeIntegrator_PrevRe_f = 0;
  }

  /* End of Update for DiscreteIntegrator: '<S6>/Discrete-Time Integrator' */

  /* Update for DiscreteIntegrator: '<S21>/Discrete-Time Integrator' incorporates:
   *  Sum: '<S21>/Add'
   */
  if (!inst->bur_HiContr_B.Input5_c) {
    inst->bur_HiContr_DWork.DiscreteTimeIntegrator_DSTATE_c += (real32_T)(((real_T)
      rtb_invert - rtb_Divide3_p) * 0.01);
    if (inst->bur_HiContr_DWork.DiscreteTimeIntegrator_DSTATE_c >= 100.0F) {
      inst->bur_HiContr_DWork.DiscreteTimeIntegrator_DSTATE_c = 100.0F;
    } else {
      if (inst->bur_HiContr_DWork.DiscreteTimeIntegrator_DSTATE_c <= 0.0F) {
        inst->bur_HiContr_DWork.DiscreteTimeIntegrator_DSTATE_c = 0.0F;
      }
    }
  }

  if (inst->bur_HiContr_B.Input5_c) {
    inst->bur_HiContr_DWork.DiscreteTimeIntegrator_PrevRe_c = 1;
  } else {
    inst->bur_HiContr_DWork.DiscreteTimeIntegrator_PrevRe_c = 0;
  }

  /* End of Update for DiscreteIntegrator: '<S21>/Discrete-Time Integrator' */

  /* Update for S-Function (sfix_udelay): '<S8>/Tapped Delay set as N_cyc!!!' */
  for (i = 0; i < 99; i++) {
    inst->bur_HiContr_DWork.TappedDelaysetasN_cyc_X[i] =
      inst->bur_HiContr_DWork.TappedDelaysetasN_cyc_X[i + 1];
  }

  inst->bur_HiContr_DWork.TappedDelaysetasN_cyc_X[99] = inst->bur_HiContr_B.Input3_g;

  /* End of Update for S-Function (sfix_udelay): '<S8>/Tapped Delay set as N_cyc!!!' */

  /* Update for DiscreteIntegrator: '<S4>/Discrete-Time Integrator' */
  if (!rtb_Compare_j) {
    inst->bur_HiContr_DWork.DiscreteTimeIntegrator_DSTATE_n += (real32_T)(0.01 * rtb_Add);
    if (inst->bur_HiContr_DWork.DiscreteTimeIntegrator_DSTATE_n >= 100.0F) {
      inst->bur_HiContr_DWork.DiscreteTimeIntegrator_DSTATE_n = 100.0F;
    } else {
      if (inst->bur_HiContr_DWork.DiscreteTimeIntegrator_DSTATE_n <= 0.0F) {
        inst->bur_HiContr_DWork.DiscreteTimeIntegrator_DSTATE_n = 0.0F;
      }
    }
  }

  if (rtb_Compare_j) {
    inst->bur_HiContr_DWork.DiscreteTimeIntegrator_PrevRe_n = 1;
  } else {
    inst->bur_HiContr_DWork.DiscreteTimeIntegrator_PrevRe_n = 0;
  }

  /* End of Update for DiscreteIntegrator: '<S4>/Discrete-Time Integrator' */
}

/* Model initialize function */
void HiContr_initialize(struct HiContr* inst)
{
  /* (no initialization code required) */
}

/* Model terminate function */
void HiContr_terminate(struct HiContr* inst)
{
  /* (no terminate code required) */
}

/*======================== TOOL VERSION INFORMATION ==========================*
 * MATLAB 8.0 (R2012b)20-Jul-2012                                             *
 * Simulink 8.0 (R2012b)20-Jul-2012                                           *
 * Simulink Coder 8.3 (R2012b)20-Jul-2012                                     *
 * Embedded Coder 6.3 (R2012b)20-Jul-2012                                     *
 * Stateflow 8.0 (R2012b)20-Jul-2012                                          *
 * Simulink Fixed Point 7.2 (R2012b)20-Jul-2012                               *
 *============================================================================*/

/*======================= LICENSE IN USE INFORMATION =========================*
 * matlab                                                                     *
 * matlab_coder                                                               *
 * real-time_workshop                                                         *
 * rtw_embedded_coder                                                         *
 * simulink                                                                   *
 *============================================================================*/
```

#### main.c
```c
/********************************************************************
 * COPYRIGHT -- Bernecker + Rainer Industrie-Elektronik Ges.m.b.H.
 ********************************************************************
 * Program: HiContr
 * File: main.c
 * Author: 106001702
 * Created: Wed Nov 09 12:46:00 2011
 ********************************************************************
 * Implementation of program HiContr
 ********************************************************************
 * Generated with B&R Automation Studio Target for Simulink V4.2
 * (ERT based)
 ********************************************************************/
#include <bur/plctypes.h>
#include "HiContr.h"
#include "rtwtypes.h"

BOOL bur_firsttime = TRUE;

/*  Defines */
#define SS_TERMINATE 4
#define SS_OUTPUT 3
#define SS_INITIALIZE 2

/*  Data Types */

/**************************** GLOBAL DATA *************************************/
/*  Definitions */

/*  Declarations  */

/***************************** FILE SCOPE DATA ********************************/

/*************************** FUNCTIONS ****************************************/
#ifdef __cplusplus

unsigned long bur_heap_size = 6553500;

#endif

void HiContr(struct HiContr* inst)
{
  switch (inst->ssMethodType)
  {
   case SS_INITIALIZE:
    /* call model initialize function */
    HiContr_initialize(inst);
    break;

   case SS_OUTPUT:
    /* call model step function */
    HiContr_step(inst);

    break;

   case SS_TERMINATE:
    /* call model terminate function */
    HiContr_terminate(inst);
    break;
  }
}

/*****************************************************************************
   Function block sample time: 0.01s
 *****************************************************************************/

/*****************************************************************************
   B&R Automation Studio Target for Simulink Version: A4.2.11 (15-Jan-2014)
 *****************************************************************************/

/*======================== TOOL VERSION INFORMATION ==========================*
 * MATLAB 8.0 (R2012b)20-Jul-2012                                             *
 * Simulink 8.0 (R2012b)20-Jul-2012                                           *
 * Simulink Coder 8.3 (R2012b)20-Jul-2012                                     *
 * Embedded Coder 6.3 (R2012b)20-Jul-2012                                     *
 * Stateflow 8.0 (R2012b)20-Jul-2012                                          *
 * Simulink Fixed Point 7.2 (R2012b)20-Jul-2012                               *
 *============================================================================*/

/*======================= LICENSE IN USE INFORMATION =========================*
 * matlab                                                                     *
 * matlab_coder                                                               *
 * real-time_workshop                                                         *
 * rtw_embedded_coder                                                         *
 * simulink                                                                   *
 *============================================================================*/
```

#### lib_properties.txt
```
For manual assignment to hardware configuration please
add the following additional include directories:

\Logical\MATLAB_includes\R2012b\

And the following additional build options:

-lm -D MODEL=HiContr -D NUMST=1 -D NCSTATES=0 -D HAVESTDIO -D ONESTEPFCN=1 -D TERMFCN=1 -D MAT_FILE=0 -D MULTI_INSTANCE_CODE=0 -D INTEGER_CODE=0 -D MT=0 -D CLASSIC_INTERFACE=0 -D TID01EQ=0
```

### Library Logical/EngineController/Lib_EC/lHiGlob (ANSIC)

#### lHiGlob.fun
```iecst
FUNCTION_BLOCK HiGlob
  VAR_INPUT
    ssMethodType: SINT;
  END_VAR  VAR_INPUT
        SkipToPowRedGain : REAL; (*Gain for skipped cylinders leading to power reduction [%Pnom/%skippedcylinder], default = 1*)
  END_VAR
  VAR_INPUT
        KPredPmaxLim : REAL; (*Gain for gobal power reduction depending on Pmax limitation [%Pnom/events*100cycles], default = 0.1*)
  END_VAR
  VAR_INPUT
        KITPmaxLim : REAL; (*Gain for global IT retardment depending on Pmax limitation [CAD/events*100cycles], default = 0.01*)
  END_VAR
  VAR_INPUT
        ZcylEng : INT; (*Number of engine cylinders, default = 20*)
  END_VAR
  VAR_INPUT
        NCylPmaxTh : INT; (*Threshold for number of cylinders being in Pmax limits before power reduction, default = 10*)
  END_VAR
  VAR_INPUT
        EngStopErrAck : BOOL := FALSE; (*Engine has stopped and errors were acknowledged on Diane*)
  END_VAR
  VAR_INPUT
        PmaxLimPowTh : REAL; (*Threshold for Pmax limitation integrator before power reduction [events/100cycles], default = 500*)
  END_VAR
  VAR_INPUT
        PmaxLimContrEn : BOOL := FALSE; (*Pmax limit control is enabled*)
  END_VAR
  VAR_INPUT
        TdownPmax : REAL; (*Integrator emptying time constant [s], default = 100*)
  END_VAR
  VAR_INPUT
        TupPmax : REAL; (*Integrator filling time constant for ignition retardment in case of Pmax limits reached, default = 1*)
  END_VAR
  VAR_INPUT
        ITPmaxLimMax : REAL; (*Max IT retardment in case of Pmax limitation [CAD], default = 5*)
  END_VAR
  VAR_INPUT
        PmaxLimReachGlob : INT; (*Number of cylinders were Pmax limit was reached*)
  END_VAR
  VAR_INPUT
        PredPmaxLimMax : REAL; (*Max power reduction in case of Pmax limitation [% of Pnom], below engine shut down, default = 50*)
  END_VAR
  VAR_INPUT
        SkipCylNr : INT; (*Number of cylinders being skipped*)
  END_VAR
  VAR_OUTPUT
        SkipCountOut : REAL; (*Skip counter output []*)
  END_VAR
  VAR_INPUT
        SkipRefRedLimMax : REAL; (*Maximum value for power reference reduction due to skip fired cylinders [%Pnom], default = 100*)
  END_VAR
  VAR_INPUT
        MaxCylSkipBefPowRed : REAL; (*Maximum percentage of skipped cylinders before power reduction starts, default = 10*)
  END_VAR
  VAR_INPUT
        MaxSkipDurBefRefRed : REAL; (*Maximum duration with skip-fired cylinders until power reduction [cycles], default = 1e4*)
  END_VAR
  VAR_INPUT
        SkipCountLimMax : REAL; (*Maximum value of skip counter [cycles], default = 1e5, must be always higher than MaxSkipDurBefRefRed*)
  END_VAR
  VAR_INPUT
        SkipRefRedLimMin : REAL; (*Minimum value for power reference reduction due to skip fired cylinders [%Pnom], default = 50*)
  END_VAR
  VAR_OUTPUT
        RefPowUpLim : REAL; (*Upper limit of reference power set in Diane [% Pnom]*)
  END_VAR
  VAR_INPUT
        PowRedCylMax : REAL; (*Maximum power reduction from all cylinders*)
  END_VAR
  VAR_INPUT
        MaxSkipDurBefStop : REAL; (*Maximum duration for overall steady skip-fired operation and reduced ref power limit until engine shut down [s], default = 1e6*)
  END_VAR
  VAR_INPUT
        SkipOvCountLimMax : REAL; (*Maximum value of overall skip-fire counter*)
  END_VAR
  VAR_INPUT
        MaxCylSkipBefStop : REAL; (*Maximum percentage of skipped cylinders before engine shut down, default = 50*)
  END_VAR
  VAR_OUTPUT
        EngShutDwn : BOOL := FALSE; (*Engine shut down command Prio 2 []*)
  END_VAR
  VAR_OUTPUT
        PowRefRedFin : REAL; (*Final global power reduction from hierarchic control [% Pnom]*)
  END_VAR
  VAR_OUTPUT
        ITGlobOffsetPmax : REAL; (*Global ignition timing retardment from Pmax controll [CAD]*)
  END_VAR
  VAR_OUTPUT
        PowRefRedGlob : REAL; (*Global power reduction from hierarchic control [% Pnom]*)
  END_VAR
  VAR_OUTPUT
        LEANOXCor : REAL; (*LEANOX correction factor due to skipfire []*)
  END_VAR
  VAR_INPUT
        TSkipCount : REAL; (*Should be 1*)
  END_VAR
  VAR_INPUT
        TSkipCount1 : REAL; (*Should be 1*)
  END_VAR
	VAR
		bur_HiGlob_DWork : D_Work_HiGlob;
	END_VAR
	VAR
		bur_HiGlob_B : BlockIO_HiGlob;
	END_VAR
END_FUNCTION_BLOCK
```

#### lHiGlob.typ
```iecst
 TYPE

END_TYPE
TYPE
	D_Work_HiGlob : STRUCT

		DiscreteTimeIntegrator_DSTATE : REAL;
		DiscreteTimeIntegrator_DSTATE_i : REAL;
		DiscreteTimeIntegrator_DSTATE_o : REAL;
		DiscreteTimeIntegrator_PrevRese : SINT;
		DiscreteTimeIntegrator_PrevRe_o : SINT;
		DiscreteTimeIntegrator_PrevRe_n : SINT;
	END_STRUCT;

	 BlockIO_HiGlob : STRUCT

		Input3 : REAL;
		Input1 : REAL;
		Input2 : REAL;
		Input4 : REAL;
		Switch2 : REAL;
		Input15 : REAL;
		Switch2_j : REAL;
		DiscreteTimeIntegrator : REAL;
		Input5 : REAL;
		Input2_f : REAL;
		Input4_i : REAL;
		Input3_a : REAL;
		Input6 : REAL;
		Switch2_d : REAL;
		Input14 : REAL;
		MinMax : REAL;
		Input9 : REAL;
		Input7 : REAL;
		Input8 : REAL;
		Divide : REAL;
		Input16 : REAL;
		Input17 : REAL;
		Input11 : INT;
		Input15_p : INT;
		Input10 : INT;
		Input1_p : INT;
		Input12 : BOOL;
		Input13 : BOOL;
		LogicalOperator : BOOL;
	END_STRUCT;

END_TYPE
```

#### HiGlob.h
```c
/********************************************************************
 * COPYRIGHT -- Bernecker + Rainer Industrie-Elektronik Ges.m.b.H.
 ********************************************************************
 * Program: HiGlob
 * File: HiGlob.h
 * Author: 106001702
 * Created: Wed Nov 09 12:46:00 2011
 ********************************************************************
 * Header for program HiGlob
 ********************************************************************
 * Generated with B&R Automation Studio Target for Simulink V4.0
 * (ERT based)
 ********************************************************************/

#ifndef RTW_HEADER_HiGlob_h_
#define RTW_HEADER_HiGlob_h_
#ifndef HiGlob_COMMON_INCLUDES_
# define HiGlob_COMMON_INCLUDES_
#include "rtwtypes.h"
#endif                                 /* HiGlob_COMMON_INCLUDES_ */

#include "HiGlob_types.h"
#include "lHiGlob.h"

/* Macros for accessing real-time model data structure */
#ifndef rtmGetErrorStatus
# define rtmGetErrorStatus(rtm)        ((void*) 0)
#endif

#ifndef rtmSetErrorStatus
# define rtmSetErrorStatus(rtm, val)   ((void) 0)
#endif

#ifndef rtmGetStopRequested
# define rtmGetStopRequested(rtm)      ((void*) 0)
#endif

#ifndef MIN
#define MIN(a,b)                       ((a) < (b) ? (a) : (b))
#endif

#ifndef MAX
#define MAX(a,b)                       ((a) > (b) ? (a) : (b))
#endif

/* Block signals (auto storage) */

/* Block states (auto storage) for system '<Root>' */

/* Block signals (auto storage) */
extern BlockIO_HiGlob HiGlob_B;

/* Block states (auto storage) */
extern D_Work_HiGlob HiGlob_DWork;

/* Model entry point functions */
extern void HiGlob_initialize(struct HiGlob* inst);
extern void HiGlob_step(struct HiGlob* inst);
extern void HiGlob_terminate(struct HiGlob* inst);

/*-
 * The generated code includes comments that allow you to trace directly
 * back to the appropriate location in the model.  The basic format
 * is <system>/block_name, where system is the system number (uniquely
 * assigned by Simulink) and block_name is the name of the block.
 *
 * Use the MATLAB hilite_system command to trace the generated code back
 * to the model.  For example,
 *
 * hilite_system('<S3>')    - opens system 3
 * hilite_system('<S3>/Kp') - opens and selects block Kp which resides in S3
 *
 * Here is the system hierarchy for this model
 *
 * '<Root>' : HiGlob
 * '<S1>'   : HiGlob/Compare To Zero
 * '<S2>'   : HiGlob/CylSkipped
 * '<S3>'   : HiGlob/Model Info
 * '<S4>'   : HiGlob/PmaxLimitGlobal
 * '<S5>'   : HiGlob/Saturation Dynamic1
 * '<S6>'   : HiGlob/Saturation Dynamic2
 * '<S7>'   : HiGlob/Saturation Dynamic3
 * '<S8>'   : HiGlob/Saturation Dynamic4
 * '<S9>'   : HiGlob/SkipCounter
 * '<S10>'  : HiGlob/SkipCounter1
 * '<S11>'  : HiGlob/threshold
 * '<S12>'  : HiGlob/threshold1
 * '<S13>'  : HiGlob/threshold2
 * '<S14>'  : HiGlob/threshold3
 * '<S15>'  : HiGlob/threshold4
 * '<S16>'  : HiGlob/PmaxLimitGlobal/Compare To threshold
 * '<S17>'  : HiGlob/PmaxLimitGlobal/PmaxLimit Integrator
 * '<S18>'  : HiGlob/PmaxLimitGlobal/Saturation Dynamic
 * '<S19>'  : HiGlob/PmaxLimitGlobal/Saturation Dynamic1
 * '<S20>'  : HiGlob/PmaxLimitGlobal/Saturation Dynamic2
 */
#endif                                 /* RTW_HEADER_HiGlob_h_ */
```

#### HiGlob_private.h
```c
/********************************************************************
 * COPYRIGHT -- Bernecker + Rainer Industrie-Elektronik Ges.m.b.H.
 ********************************************************************
 * Program: HiGlob
 * File: HiGlob_private.h
 * Author: 106001702
 * Created: Wed Nov 09 12:46:00 2011
 ********************************************************************
 * Header for program HiGlob
 ********************************************************************
 * Generated with B&R Automation Studio Target for Simulink V4.0
 * (ERT based)
 ********************************************************************/

#ifndef RTW_HEADER_HiGlob_private_h_
#define RTW_HEADER_HiGlob_private_h_
#include "rtwtypes.h"
#include <bur/plctypes.h>
#ifndef __RTWTYPES_H__
#error This file requires rtwtypes.h to be included
#else
#ifdef TMWTYPES_PREVIOUSLY_INCLUDED
#error This file requires rtwtypes.h to be included before tmwtypes.h
#else

/* Check for inclusion of an incorrect version of rtwtypes.h */
#ifndef RTWTYPES_ID_C08S16I32L32N32F1
#error This code was generated with a different "rtwtypes.h" than the file included
#endif                                 /* RTWTYPES_ID_C08S16I32L32N32F1 */
#endif                                 /* TMWTYPES_PREVIOUSLY_INCLUDED */
#endif                                 /* __RTWTYPES_H__ */

#ifndef MIN
#define MIN(a,b)                       ((a) < (b) ? (a) : (b))
#endif

#ifndef MAX
#define MAX(a,b)                       ((a) > (b) ? (a) : (b))
#endif

/* Imported (extern) block parameters */
extern real32_T KITPmaxLim;            /* Variable: KITPmaxLim
                                        * Referenced by: '<S4>/KITPmaxLim (CAD//events*100cycles)'
                                        */
extern real32_T KPredPmaxLim;          /* Variable: KPredPmaxLim
                                        * Referenced by: '<S4>/KPredPmaxLim (%Pel//events*100cycles)'
                                        */
extern real32_T SkipToPowRedGain;      /* Variable: SkipToPowRedGain
                                        * Referenced by: '<Root>/SkipToPowRedGain'
                                        */

#endif                                 /* RTW_HEADER_HiGlob_private_h_ */
```

#### HiGlob_types.h
```c
/********************************************************************
 * COPYRIGHT -- Bernecker + Rainer Industrie-Elektronik Ges.m.b.H.
 ********************************************************************
 * Program: HiGlob
 * File: HiGlob_types.h
 * Author: 106001702
 * Created: Wed Nov 09 12:46:00 2011
 ********************************************************************
 * Header for program HiGlob
 ********************************************************************
 * Generated with B&R Automation Studio Target for Simulink V4.0
 * (ERT based)
 ********************************************************************/

#ifndef RTW_HEADER_HiGlob_types_h_
#define RTW_HEADER_HiGlob_types_h_
#ifndef MIN
#define MIN(a,b)                       ((a) < (b) ? (a) : (b))
#endif

#ifndef MAX
#define MAX(a,b)                       ((a) > (b) ? (a) : (b))
#endif
#endif                                 /* RTW_HEADER_HiGlob_types_h_ */
```

#### rtwtypes.h
```c
/********************************************************************
 * COPYRIGHT -- Bernecker + Rainer Industrie-Elektronik Ges.m.b.H.
 ********************************************************************
 * Program: HiGlob
 * File: rtwtypes.h
 * Author: 106001702
 * Created: Wed Nov 09 12:46:00 2011
 ********************************************************************
 * Header for program HiGlob
 ********************************************************************
 * Generated with B&R Automation Studio Target for Simulink V4.0
 * (ERT based)
 ********************************************************************/

#ifndef RTW_HEADER_rtwtypes_h_
#define RTW_HEADER_rtwtypes_h_
#ifndef __RTWTYPES_H__
#define __RTWTYPES_H__
#ifndef TRUE
# define TRUE                          (1U)
#endif

#ifndef FALSE
# define FALSE                         (0U)
#endif

#ifndef __TMWTYPES__
#define __TMWTYPES__
#include <limits.h>

/*=======================================================================*
 * Target hardware information
 *   Device type: Intel->x86/Pentium
 *   Number of bits:     char:   8    short:   16    int:  32
 *                       long:  32      native word size:  32
 *   Byte ordering: LittleEndian
 *   Signed integer division rounds to: Zero
 *   Shift right on a signed integer as arithmetic shift: on
 *=======================================================================*/

/*=======================================================================*
 * Fixed width word size data types:                                     *
 *   int8_T, int16_T, int32_T     - signed 8, 16, or 32 bit integers     *
 *   uint8_T, uint16_T, uint32_T  - unsigned 8, 16, or 32 bit integers   *
 *   real32_T, real64_T           - 32 and 64 bit floating point numbers *
 *=======================================================================*/
typedef signed char int8_T;
typedef unsigned char uint8_T;
typedef short int16_T;
typedef unsigned short uint16_T;
typedef int int32_T;
typedef unsigned int uint32_T;
typedef float real32_T;
typedef double real64_T;

/*===========================================================================*
 * Generic type definitions: real_T, time_T, boolean_T, int_T, uint_T,       *
 *                           ulong_T, char_T and byte_T.                     *
 *===========================================================================*/
typedef double real_T;
typedef double time_T;
typedef unsigned char boolean_T;
typedef int int_T;
typedef unsigned int uint_T;
typedef unsigned long ulong_T;
typedef char char_T;
typedef unsigned char uchar_T;
typedef char_T byte_T;

/*=======================================================================*
 * Min and Max:                                                          *
 *   int8_T, int16_T, int32_T     - signed 8, 16, or 32 bit integers     *
 *   uint8_T, uint16_T, uint32_T  - unsigned 8, 16, or 32 bit integers   *
 *=======================================================================*/
#define MAX_int8_T                     ((int8_T)(127))
#define MIN_int8_T                     ((int8_T)(-128))
#define MAX_uint8_T                    ((uint8_T)(255U))
#define MIN_uint8_T                    ((uint8_T)(0U))
#define MAX_int16_T                    ((int16_T)(32767))
#define MIN_int16_T                    ((int16_T)(-32768))
#define MAX_uint16_T                   ((uint16_T)(65535U))
#define MIN_uint16_T                   ((uint16_T)(0U))
#define MAX_int32_T                    ((int32_T)(2147483647))
#define MIN_int32_T                    ((int32_T)(-2147483647-1))
#define MAX_uint32_T                   ((uint32_T)(0xFFFFFFFFU))
#define MIN_uint32_T                   ((uint32_T)(0U))

/* Logical type definitions */
#if (!defined(__cplusplus)) && (!defined(__true_false_are_keywords))
#  ifndef false
#   define false                       (0U)
#  endif

#  ifndef true
#   define true                        (1U)
#  endif
#endif

/*
 * Simulink Coder assumes the code is compiled on a target using a 2's complement representation
 * for signed integer values.
 */
#if ((SCHAR_MIN + 1) != -SCHAR_MAX)
#error "This code must be compiled using a 2's complement representation for signed integer values"
#endif

/* This ID is used to detect inclusion of an incompatible rtwtypes.h */
#define RTWTYPES_ID_C08S16I32L32N32F1
#else                                  /* __TMWTYPES__ */
#define TMWTYPES_PREVIOUSLY_INCLUDED
#endif                                 /* __TMWTYPES__ */

/* Block D-Work pointer type */
typedef void * pointer_T;

/* Simulink specific types */
#ifndef __SIMSTRUC_TYPES_H__
#define __SIMSTRUC_TYPES_H__

/* Trigger directions: falling, either, and rising */
typedef enum {
  FALLING_ZERO_CROSSING = -1,
  ANY_ZERO_CROSSING = 0,
  RISING_ZERO_CROSSING = 1
} ZCDirection;

/* Previous state of a trigger signal */
typedef uint8_T ZCSigState;

/* Initial value of a trigger zero crossing signal */
#define UNINITIALIZED_ZCSIG            0x03U
#define NEG_ZCSIG                      0x02U
#define POS_ZCSIG                      0x01U
#define ZERO_ZCSIG                     0x00U

/* Current state of a trigger signal */
typedef enum {
  FALLING_ZCEVENT = -1,
  NO_ZCEVENT = 0,
  RISING_ZCEVENT = 1
} ZCEventType;

#endif                                 /* __SIMSTRUC_TYPES_H__ */
#endif                                 /* __RTWTYPES_H__ */

#ifndef MIN
#define MIN(a,b)                       ((a) < (b) ? (a) : (b))
#endif

#ifndef MAX
#define MAX(a,b)                       ((a) > (b) ? (a) : (b))
#endif
#endif                                 /* RTW_HEADER_rtwtypes_h_ */
```

#### HiGlob.c
```c
/********************************************************************
 * COPYRIGHT -- Bernecker + Rainer Industrie-Elektronik Ges.m.b.H.
 ********************************************************************
 * Program: HiGlob
 * File: HiGlob.c
 * Author: 106001702
 * Created: Wed Nov 09 12:46:00 2011
 ********************************************************************
 * Implementation of program HiGlob
 ********************************************************************
 * Generated with B&R Automation Studio Target for Simulink V4.0
 * (ERT based)
 ********************************************************************/

#include "HiGlob.h"
#include "HiGlob_private.h"

/*  Defines */

/*  Data Types */

/**************************** GLOBAL DATA *************************************/
/*  Definitions */

/* Block signals (auto storage) */

/* Block states (auto storage) */

/*  Declarations  */

/***************************** FILE SCOPE DATA ********************************/

/*************************** FUNCTIONS ****************************************/

/* Model step function */
void HiGlob_step(struct HiGlob* inst)
{
  /* local block i/o variables */
  boolean_T rtb_BitwiseOperator;
  boolean_T rtb_BitwiseOperator1;
  real32_T rtb_MinMax2;
  real32_T rtb_percent;
  real32_T rtb_Divide_n;
  real_T rtb_Divide;
  int16_T rtb_Subtract1;
  boolean_T rtb_LowerRelop1_l;
  boolean_T rtb_Compare_jf;
  int16_T rtb_Switch_o;

  /* S-Function (bur_in): '<Root>/Input11' */
  inst->bur_HiGlob_B.Input11 = inst->ZcylEng;

  /* S-Function (bur_in): '<S4>/Input15' */
  inst->bur_HiGlob_B.Input15_p = inst->NCylPmaxTh;

  /* Sum: '<S4>/Add' */
  rtb_Switch_o = (int16_T)(inst->bur_HiGlob_B.Input11 - inst->bur_HiGlob_B.Input15_p);

  /* S-Function (bur_in): '<Root>/Input12' */
  inst->bur_HiGlob_B.Input12 = inst->EngStopErrAck;

  /* DiscreteIntegrator: '<S17>/Discrete-Time Integrator' */
  if (inst->bur_HiGlob_B.Input12 || (inst->bur_HiGlob_DWork.DiscreteTimeIntegrator_PrevRese != 0)) {
    inst->bur_HiGlob_DWork.DiscreteTimeIntegrator_DSTATE = 0.0F;
  }

  if (inst->bur_HiGlob_DWork.DiscreteTimeIntegrator_DSTATE >= 1000.0F) {
    inst->bur_HiGlob_DWork.DiscreteTimeIntegrator_DSTATE = 1000.0F;
  } else {
    if (inst->bur_HiGlob_DWork.DiscreteTimeIntegrator_DSTATE <= 0.0F) {
      inst->bur_HiGlob_DWork.DiscreteTimeIntegrator_DSTATE = 0.0F;
    }
  }

  rtb_MinMax2 = inst->bur_HiGlob_DWork.DiscreteTimeIntegrator_DSTATE;

  /* End of DiscreteIntegrator: '<S17>/Discrete-Time Integrator' */

  /* S-Function (bur_in): '<S4>/Input3' */
  inst->bur_HiGlob_B.Input3 = inst->PmaxLimPowTh;

  /* Sum: '<S4>/Add1' */
  rtb_percent = rtb_MinMax2 - inst->bur_HiGlob_B.Input3;

  /* Gain: '<S4>/KITPmaxLim (CAD//events*100cycles)' */
  rtb_MinMax2 *= inst->KITPmaxLim;

  /* S-Function (bur_in): '<Root>/Input13' */
  inst->bur_HiGlob_B.Input13 = inst->PmaxLimContrEn;

  /* Product: '<S4>/Divide' */
  rtb_Divide_n = inst->bur_HiGlob_B.Input13 ? rtb_MinMax2 : 0.0F;

  /* S-Function (bur_in): '<S4>/Input1' */
  inst->bur_HiGlob_B.Input1 = inst->TdownPmax;

  /* S-Function (bur_in): '<S4>/Input2' */
  inst->bur_HiGlob_B.Input2 = inst->TupPmax;

  /* S-Function (bur_in): '<S4>/Input4' */
  inst->bur_HiGlob_B.Input4 = inst->ITPmaxLimMax;

  /* Switch: '<S4>/Switch3' incorporates:
   *  Constant: '<S16>/Constant'
   *  Constant: '<S4>/Constant4'
   *  Logic: '<S4>/Logical Operator13'
   *  RelationalOperator: '<S16>/Compare'
   */
  if (!((rtb_percent > 0.0F) && inst->bur_HiGlob_B.Input13)) {
    rtb_percent = 0.0F;
  }

  /* End of Switch: '<S4>/Switch3' */

  /* Gain: '<S4>/KPredPmaxLim (%Pel//events*100cycles)' */
  rtb_MinMax2 = inst->KPredPmaxLim * rtb_percent;

  /* Product: '<S17>/Divide1' incorporates:
   *  Constant: '<S17>/Constant'
   */
  rtb_Divide = 1.0 / (real_T)inst->bur_HiGlob_B.Input1;

  /* S-Function (bur_in): '<Root>/Input10' */
  inst->bur_HiGlob_B.Input10 = inst->PmaxLimReachGlob;

  /* Sum: '<S4>/Subtract1' */
  rtb_Subtract1 = (int16_T)(inst->bur_HiGlob_B.Input10 - inst->bur_HiGlob_B.Input15_p);

  /* Switch: '<S18>/Switch2' incorporates:
   *  RelationalOperator: '<S18>/LowerRelop1'
   */
  if (!(rtb_Subtract1 > rtb_Switch_o)) {
    /* Switch: '<S18>/Switch' incorporates:
     *  Constant: '<S4>/Constant1'
     *  RelationalOperator: '<S18>/UpperRelop'
     */
    if (rtb_Subtract1 < 0) {
      rtb_Subtract1 = 0;
    }

    /* End of Switch: '<S18>/Switch' */
    rtb_Switch_o = rtb_Subtract1;
  }

  /* End of Switch: '<S18>/Switch2' */

  /* Product: '<S17>/Divide2' incorporates:
   *  Product: '<S17>/Divide'
   *  Sum: '<S17>/Add'
   */
  rtb_Divide = (real_T)((real32_T)rtb_Switch_o / inst->bur_HiGlob_B.Input2) - rtb_Divide;

  /* Switch: '<S19>/Switch2' incorporates:
   *  RelationalOperator: '<S19>/LowerRelop1'
   */
  if (rtb_Divide_n > inst->bur_HiGlob_B.Input4) {
    inst->bur_HiGlob_B.Switch2 = inst->bur_HiGlob_B.Input4;
  } else {
    /* Switch: '<S19>/Switch' incorporates:
     *  Constant: '<S4>/Constant6'
     *  RelationalOperator: '<S19>/UpperRelop'
     */
    if (rtb_Divide_n < 0.0F) {
      inst->bur_HiGlob_B.Switch2 = 0.0F;
    } else {
      inst->bur_HiGlob_B.Switch2 = rtb_Divide_n;
    }

    /* End of Switch: '<S19>/Switch' */
  }

  /* End of Switch: '<S19>/Switch2' */

  /* S-Function (bur_in): '<Root>/Input15' */
  inst->bur_HiGlob_B.Input15 = inst->PredPmaxLimMax;

  /* Switch: '<S20>/Switch2' incorporates:
   *  RelationalOperator: '<S20>/LowerRelop1'
   */
  if (rtb_MinMax2 > inst->bur_HiGlob_B.Input15) {
    inst->bur_HiGlob_B.Switch2_j = inst->bur_HiGlob_B.Input15;
  } else {
    /* Switch: '<S20>/Switch' incorporates:
     *  Constant: '<S4>/Constant9'
     *  RelationalOperator: '<S20>/UpperRelop'
     */
    if (rtb_MinMax2 < 0.0F) {
      inst->bur_HiGlob_B.Switch2_j = 0.0F;
    } else {
      inst->bur_HiGlob_B.Switch2_j = rtb_MinMax2;
    }

    /* End of Switch: '<S20>/Switch' */
  }

  /* End of Switch: '<S20>/Switch2' */

  /* S-Function (bur_in): '<Root>/Input1' */
  inst->bur_HiGlob_B.Input1_p = inst->SkipCylNr;

  /* Gain: '<Root>/percent' incorporates:
   *  Product: '<Root>/Divide1'
   */
  rtb_percent = (real32_T)inst->bur_HiGlob_B.Input1_p / (real32_T)inst->bur_HiGlob_B.Input11 *
    100.0F;

  /* S-Function (sfix_bitop): '<Root>/Bitwise Operator' incorporates:
   *  Constant: '<S2>/Constant'
   *  RelationalOperator: '<S2>/Compare'
   */
  rtb_BitwiseOperator = !(rtb_percent > 0.0F);

  /* DiscreteIntegrator: '<S9>/Discrete-Time Integrator' */
  if (rtb_BitwiseOperator || (inst->bur_HiGlob_DWork.DiscreteTimeIntegrator_PrevRe_o != 0))
  {
    inst->bur_HiGlob_DWork.DiscreteTimeIntegrator_DSTATE_i = 0.0F;
  }

  if (inst->bur_HiGlob_DWork.DiscreteTimeIntegrator_DSTATE_i >= 1.0E+6F) {
    inst->bur_HiGlob_DWork.DiscreteTimeIntegrator_DSTATE_i = 1.0E+6F;
  } else {
    if (inst->bur_HiGlob_DWork.DiscreteTimeIntegrator_DSTATE_i <= 0.0F) {
      inst->bur_HiGlob_DWork.DiscreteTimeIntegrator_DSTATE_i = 0.0F;
    }
  }

  inst->bur_HiGlob_B.DiscreteTimeIntegrator = inst->bur_HiGlob_DWork.DiscreteTimeIntegrator_DSTATE_i;

  /* End of DiscreteIntegrator: '<S9>/Discrete-Time Integrator' */

  /* S-Function (bur_out): '<Root>/Output1' */
  inst->SkipCountOut = inst->bur_HiGlob_B.DiscreteTimeIntegrator;

  /* S-Function (bur_in): '<Root>/Input5' */
  inst->bur_HiGlob_B.Input5 = inst->SkipRefRedLimMax;

  /* S-Function (bur_in): '<Root>/Input2' */
  inst->bur_HiGlob_B.Input2_f = inst->MaxCylSkipBefPowRed;

  /* Sum: '<Root>/Add2' */
  rtb_MinMax2 = rtb_percent - inst->bur_HiGlob_B.Input2_f;

  /* Switch: '<Root>/Switch2' incorporates:
   *  Constant: '<Root>/Constant2'
   *  Constant: '<S11>/Constant'
   *  RelationalOperator: '<S11>/Compare'
   */
  if (!(rtb_MinMax2 > 0.0F)) {
    rtb_MinMax2 = 0.0F;
  }

  /* End of Switch: '<Root>/Switch2' */

  /* S-Function (bur_in): '<Root>/Input4' */
  inst->bur_HiGlob_B.Input4_i = inst->MaxSkipDurBefRefRed;

  /* S-Function (bur_in): '<Root>/Input3' */
  inst->bur_HiGlob_B.Input3_a = inst->SkipCountLimMax;

  /* Switch: '<S7>/Switch2' incorporates:
   *  RelationalOperator: '<S7>/LowerRelop1'
   */
  if (inst->bur_HiGlob_B.DiscreteTimeIntegrator > inst->bur_HiGlob_B.Input3_a) {
    rtb_Divide_n = inst->bur_HiGlob_B.Input3_a;
  } else {
    /* Switch: '<S7>/Switch' incorporates:
     *  Constant: '<Root>/Constant7'
     *  RelationalOperator: '<S7>/UpperRelop'
     */
    if (inst->bur_HiGlob_B.DiscreteTimeIntegrator < 0.0F) {
      rtb_Divide_n = 0.0F;
    } else {
      rtb_Divide_n = inst->bur_HiGlob_B.DiscreteTimeIntegrator;
    }

    /* End of Switch: '<S7>/Switch' */
  }

  /* End of Switch: '<S7>/Switch2' */

  /* Switch: '<Root>/Switch1' incorporates:
   *  Constant: '<Root>/Constant8'
   *  Constant: '<S12>/Constant'
   *  RelationalOperator: '<S12>/Compare'
   *  Sum: '<Root>/Add4'
   */
  if (rtb_Divide_n - inst->bur_HiGlob_B.Input4_i > 0.0F) {
    rtb_Divide_n = rtb_percent;
  } else {
    rtb_Divide_n = 0.0F;
  }

  /* End of Switch: '<Root>/Switch1' */

  /* MinMax: '<Root>/MinMax2' */
  rtb_MinMax2 = rtb_MinMax2 >= rtb_Divide_n ? rtb_MinMax2 : rtb_Divide_n;

  /* Sum: '<Root>/Add3' incorporates:
   *  Constant: '<Root>/Constant4'
   *  Gain: '<Root>/SkipToPowRedGain'
   *  MinMax: '<Root>/MinMax2'
   */
  rtb_Divide_n = 100.0F - inst->SkipToPowRedGain * rtb_MinMax2;

  /* RelationalOperator: '<S5>/LowerRelop1' */
  rtb_LowerRelop1_l = (rtb_Divide_n > inst->bur_HiGlob_B.Input5);

  /* S-Function (bur_in): '<Root>/Input6' */
  inst->bur_HiGlob_B.Input6 = inst->SkipRefRedLimMin;

  /* Switch: '<S5>/Switch2' */
  if (rtb_LowerRelop1_l) {
    inst->bur_HiGlob_B.Switch2_d = inst->bur_HiGlob_B.Input5;
  } else {
    /* Switch: '<S5>/Switch' incorporates:
     *  RelationalOperator: '<S5>/UpperRelop'
     */
    if (rtb_Divide_n < inst->bur_HiGlob_B.Input6) {
      inst->bur_HiGlob_B.Switch2_d = inst->bur_HiGlob_B.Input6;
    } else {
      inst->bur_HiGlob_B.Switch2_d = rtb_Divide_n;
    }

    /* End of Switch: '<S5>/Switch' */
  }

  /* End of Switch: '<S5>/Switch2' */

  /* S-Function (bur_out): '<Root>/Output2' */
  inst->RefPowUpLim = inst->bur_HiGlob_B.Switch2_d;

  /* S-Function (bur_in): '<Root>/Input14' */
  inst->bur_HiGlob_B.Input14 = inst->PowRedCylMax;

  /* MinMax: '<Root>/MinMax' */
  inst->bur_HiGlob_B.MinMax = inst->bur_HiGlob_B.Input14 >= inst->bur_HiGlob_B.Switch2_j ? inst->bur_HiGlob_B.Input14 :
    inst->bur_HiGlob_B.Switch2_j;

  /* RelationalOperator: '<S15>/Compare' incorporates:
   *  Constant: '<S15>/Constant'
   *  Sum: '<Root>/Add7'
   */
  rtb_LowerRelop1_l = (inst->bur_HiGlob_B.MinMax - inst->bur_HiGlob_B.Input15 > 0.0F);

  /* S-Function (bur_in): '<Root>/Input9' */
  inst->bur_HiGlob_B.Input9 = inst->MaxSkipDurBefStop;

  /* S-Function (bur_in): '<Root>/Input7' */
  inst->bur_HiGlob_B.Input7 = inst->SkipOvCountLimMax;

  /* S-Function (sfix_bitop): '<Root>/Bitwise Operator1' incorporates:
   *  Constant: '<S1>/Constant'
   *  MinMax: '<Root>/MinMax2'
   *  RelationalOperator: '<S1>/Compare'
   */
  rtb_BitwiseOperator1 = !(rtb_MinMax2 > 0.0F);

  /* DiscreteIntegrator: '<S10>/Discrete-Time Integrator' */
  if (rtb_BitwiseOperator1 || (inst->bur_HiGlob_DWork.DiscreteTimeIntegrator_PrevRe_n != 0))
  {
    inst->bur_HiGlob_DWork.DiscreteTimeIntegrator_DSTATE_o = 0.0F;
  }

  if (inst->bur_HiGlob_DWork.DiscreteTimeIntegrator_DSTATE_o >= 1.0E+7F) {
    inst->bur_HiGlob_DWork.DiscreteTimeIntegrator_DSTATE_o = 1.0E+7F;
  } else {
    if (inst->bur_HiGlob_DWork.DiscreteTimeIntegrator_DSTATE_o <= 0.0F) {
      inst->bur_HiGlob_DWork.DiscreteTimeIntegrator_DSTATE_o = 0.0F;
    }
  }

  /* End of DiscreteIntegrator: '<S10>/Discrete-Time Integrator' */

  /* Switch: '<S8>/Switch2' incorporates:
   *  DiscreteIntegrator: '<S10>/Discrete-Time Integrator'
   *  RelationalOperator: '<S8>/LowerRelop1'
   */
  if (inst->bur_HiGlob_DWork.DiscreteTimeIntegrator_DSTATE_o > inst->bur_HiGlob_B.Input7) {
    rtb_Divide_n = inst->bur_HiGlob_B.Input7;
  } else {
    /* Switch: '<S8>/Switch' incorporates:
     *  Constant: '<Root>/Constant11'
     *  RelationalOperator: '<S8>/UpperRelop'
     */
    if ((real_T)inst->bur_HiGlob_DWork.DiscreteTimeIntegrator_DSTATE_o < 0.0) {
      rtb_Divide_n = 0.0F;
    } else {
      rtb_Divide_n = inst->bur_HiGlob_DWork.DiscreteTimeIntegrator_DSTATE_o;
    }

    /* End of Switch: '<S8>/Switch' */
  }

  /* End of Switch: '<S8>/Switch2' */

  /* RelationalOperator: '<S14>/Compare' incorporates:
   *  Constant: '<S14>/Constant'
   *  Sum: '<Root>/Add6'
   */
  rtb_Compare_jf = (rtb_Divide_n - inst->bur_HiGlob_B.Input9 > 0.0F);

  /* S-Function (bur_in): '<Root>/Input8' */
  inst->bur_HiGlob_B.Input8 = inst->MaxCylSkipBefStop;

  /* Logic: '<Root>/Logical Operator' incorporates:
   *  Constant: '<S13>/Constant'
   *  RelationalOperator: '<S13>/Compare'
   *  Sum: '<Root>/Add5'
   */
  inst->bur_HiGlob_B.LogicalOperator = ((rtb_LowerRelop1_l || rtb_Compare_jf ||
    (rtb_percent - inst->bur_HiGlob_B.Input8 > 0.0F)));

  /* S-Function (bur_out): '<Root>/Output3' */
  inst->EngShutDwn = inst->bur_HiGlob_B.LogicalOperator;

  /* S-Function (bur_out): '<Root>/Output4' */
  inst->PowRefRedFin = inst->bur_HiGlob_B.MinMax;

  /* S-Function (bur_out): '<Root>/Output5' */
  inst->ITGlobOffsetPmax = inst->bur_HiGlob_B.Switch2;

  /* S-Function (bur_out): '<Root>/Output6' */
  inst->PowRefRedGlob = inst->bur_HiGlob_B.Switch2_j;

  /* Sum: '<Root>/Add1' incorporates:
   *  Constant: '<Root>/Constant'
   */
  rtb_Switch_o = (int16_T)(inst->bur_HiGlob_B.Input11 - 1);

  /* Switch: '<S6>/Switch2' incorporates:
   *  RelationalOperator: '<S6>/LowerRelop1'
   */
  if (!(inst->bur_HiGlob_B.Input1_p > rtb_Switch_o)) {
    /* Switch: '<S6>/Switch' incorporates:
     *  Constant: '<Root>/Constant1'
     *  RelationalOperator: '<S6>/UpperRelop'
     */
    if (inst->bur_HiGlob_B.Input1_p < 0) {
      rtb_Switch_o = 0;
    } else {
      rtb_Switch_o = inst->bur_HiGlob_B.Input1_p;
    }

    /* End of Switch: '<S6>/Switch' */
  }

  /* End of Switch: '<S6>/Switch2' */

  /* Sum: '<Root>/Add' */
  rtb_Switch_o = (int16_T)(inst->bur_HiGlob_B.Input11 - rtb_Switch_o);

  /* Product: '<Root>/Divide' */
  inst->bur_HiGlob_B.Divide = (real32_T)inst->bur_HiGlob_B.Input11 / (real32_T)rtb_Switch_o;

  /* S-Function (bur_out): '<Root>/Output9' */
  inst->LEANOXCor = inst->bur_HiGlob_B.Divide;

  /* S-Function (bur_in): '<Root>/Input16' */
  inst->bur_HiGlob_B.Input16 = inst->TSkipCount;

  /* S-Function (bur_in): '<Root>/Input17' */
  inst->bur_HiGlob_B.Input17 = inst->TSkipCount1;

  /* Update for DiscreteIntegrator: '<S17>/Discrete-Time Integrator' */
  if (!inst->bur_HiGlob_B.Input12) {
    inst->bur_HiGlob_DWork.DiscreteTimeIntegrator_DSTATE = (real32_T)(0.01 * rtb_Divide) +
      inst->bur_HiGlob_DWork.DiscreteTimeIntegrator_DSTATE;
    if (inst->bur_HiGlob_DWork.DiscreteTimeIntegrator_DSTATE >= 1000.0F) {
      inst->bur_HiGlob_DWork.DiscreteTimeIntegrator_DSTATE = 1000.0F;
    } else {
      if (inst->bur_HiGlob_DWork.DiscreteTimeIntegrator_DSTATE <= 0.0F) {
        inst->bur_HiGlob_DWork.DiscreteTimeIntegrator_DSTATE = 0.0F;
      }
    }
  }

  if (inst->bur_HiGlob_B.Input12) {
    inst->bur_HiGlob_DWork.DiscreteTimeIntegrator_PrevRese = 1;
  } else {
    inst->bur_HiGlob_DWork.DiscreteTimeIntegrator_PrevRese = 0;
  }

  /* End of DiscreteIntegrator: '<S17>/Discrete-Time Integrator' */

  /* Update for DiscreteIntegrator: '<S9>/Discrete-Time Integrator' */
  if (!rtb_BitwiseOperator) {
    if (inst->bur_HiGlob_DWork.DiscreteTimeIntegrator_DSTATE_i >= 1.0E+6F) {
      inst->bur_HiGlob_DWork.DiscreteTimeIntegrator_DSTATE_i = 1.0E+6F;
    } else {
      if (inst->bur_HiGlob_DWork.DiscreteTimeIntegrator_DSTATE_i <= 0.0F) {
        inst->bur_HiGlob_DWork.DiscreteTimeIntegrator_DSTATE_i = 0.0F;
      }
    }
  }

  if (rtb_BitwiseOperator) {
    inst->bur_HiGlob_DWork.DiscreteTimeIntegrator_PrevRe_o = 1;
  } else {
    inst->bur_HiGlob_DWork.DiscreteTimeIntegrator_PrevRe_o = 0;
  }

  /* End of DiscreteIntegrator: '<S9>/Discrete-Time Integrator' */

  /* Update for DiscreteIntegrator: '<S10>/Discrete-Time Integrator' */
  if (!rtb_BitwiseOperator1) {
    if (inst->bur_HiGlob_DWork.DiscreteTimeIntegrator_DSTATE_o >= 1.0E+7F) {
      inst->bur_HiGlob_DWork.DiscreteTimeIntegrator_DSTATE_o = 1.0E+7F;
    } else {
      if (inst->bur_HiGlob_DWork.DiscreteTimeIntegrator_DSTATE_o <= 0.0F) {
        inst->bur_HiGlob_DWork.DiscreteTimeIntegrator_DSTATE_o = 0.0F;
      }
    }
  }

  if (rtb_BitwiseOperator1) {
    inst->bur_HiGlob_DWork.DiscreteTimeIntegrator_PrevRe_n = 1;
  } else {
    inst->bur_HiGlob_DWork.DiscreteTimeIntegrator_PrevRe_n = 0;
  }

  /* End of DiscreteIntegrator: '<S10>/Discrete-Time Integrator' */
}

/* Model initialize function */
void HiGlob_initialize(struct HiGlob* inst)
{
  /* (no initialization code required) */
}

/* Model terminate function */
void HiGlob_terminate(struct HiGlob* inst)
{
  /* (no terminate code required) */
}

/*======================== TOOL VERSION INFORMATION ==========================*
 * MATLAB 7.12 (R2011a)09-Mar-2011                                            *
 * Simulink 7.7 (R2011a)09-Mar-2011                                           *
 * Simulink Coder 8.0 (R2011a)09-Mar-2011                                     *
 * Embedded Coder 6.0 (R2011a)09-Mar-2011                                     *
 * Stateflow 7.7 (R2011a)09-Mar-2011                                          *
 * Simulink Fixed Point 6.5 (R2011a)09-Mar-2011                               *
 *============================================================================*/

/*======================= LICENSE IN USE INFORMATION =========================*
 * matlab                                                                     *
 * matlab_coder                                                               *
 * real-time_workshop                                                         *
 * rtw_embedded_coder                                                         *
 * simulink                                                                   *
 *============================================================================*/
```

#### main.c
```c
/********************************************************************
 * COPYRIGHT -- Bernecker + Rainer Industrie-Elektronik Ges.m.b.H.
 ********************************************************************
 * Program: HiGlob
 * File: main.c
 * Author: 106001702
 * Created: Wed Nov 09 12:46:00 2011
 ********************************************************************
 * Implementation of program HiGlob
 ********************************************************************
 * Generated with B&R Automation Studio Target for Simulink V4.0
 * (ERT based)
 ********************************************************************/

#include <bur/plctypes.h>
#include "HiGlob.h"
#include "rtwtypes.h"

BOOL bur_firsttime = TRUE;

/*  Defines */
#define SS_TERMINATE 4
#define SS_OUTPUT 3
#define SS_INITIALIZE 2

/*  Data Types */

/**************************** GLOBAL DATA *************************************/
/*  Definitions */

/*  Declarations  */

/***************************** FILE SCOPE DATA ********************************/

/*************************** FUNCTIONS ****************************************/
#ifdef __cplusplus

unsigned long bur_heap_size = 65535;

#endif

void HiGlob(struct HiGlob* inst)
{
  switch (inst->ssMethodType)
  {
   case SS_INITIALIZE:
    /* call model initialize function */
    HiGlob_initialize(inst);
    break;

   case SS_OUTPUT:
    /* call model step function */
    HiGlob_step(inst);

    break;

   case SS_TERMINATE:
    /* call model terminate function */
    HiGlob_terminate(inst);
    break;
  }
}

/*****************************************************************************
   Function block sample time: 0.01s
 *****************************************************************************/

/*****************************************************************************
   B&R Automation Studio Target for Simulink Version: A4.0.48 (27-Jun-2013)
 *****************************************************************************/

/*======================== TOOL VERSION INFORMATION ==========================*
 * MATLAB 7.12 (R2011a)09-Mar-2011                                            *
 * Simulink 7.7 (R2011a)09-Mar-2011                                           *
 * Simulink Coder 8.0 (R2011a)09-Mar-2011                                     *
 * Embedded Coder 6.0 (R2011a)09-Mar-2011                                     *
 * Stateflow 7.7 (R2011a)09-Mar-2011                                          *
 * Simulink Fixed Point 6.5 (R2011a)09-Mar-2011                               *
 *============================================================================*/

/*======================= LICENSE IN USE INFORMATION =========================*
 * matlab                                                                     *
 * matlab_coder                                                               *
 * real-time_workshop                                                         *
 * rtw_embedded_coder                                                         *
 * simulink                                                                   *
 *============================================================================*/
```

#### lib_properties.txt
```
For manual assignment to hardware configuration please
add the following additional include directories:

\Logical\MATLAB_includes\R2011a\

And the following additional build options:

-lm -D MODEL=HiGlob -D NUMST=1 -D NCSTATES=0 -D HAVESTDIO -D ONESTEPFCN=1 -D TERMFCN=1 -D MAT_FILE=0 -D MULTI_INSTANCE_CODE=0 -D INTEGER_CODE=0 -D MT=0 -D TID01EQ=0
```

### Library Logical/EngineController/Lib_EC/lMFB50Cont (ANSIC)

#### lMFB50Cont.fun
```iecst
FUNCTION_BLOCK MFB50Contr
  VAR_INPUT
    ssMethodType: SINT;
  END_VAR  VAR_INPUT
        MapPoP2sx : ARRAY[0..1] OF LREAL := [2(1000.0000000000)]; (*p2s values for map in [mbar]*)
  END_VAR
  VAR_INPUT
        MFB50GlobRefExt : LREAL := 5.0000000000; (*Global reference for MFB50 in [CADafTDC]*)
  END_VAR
  VAR_INPUT
        MFB50MedianEn : BOOL := FALSE; (*Switch to decide between different MFB50 references [boolean], 0 = global reference, 1 = median *)
  END_VAR
  VAR_INPUT
        MapPoP2sy : ARRAY[0..1] OF LREAL := [2(0.5000000000)]; (*proportional gain values for map in [CADbfTDC / CADafTDC]*)
  END_VAR
  VAR_INPUT
        MapIoP2sx : ARRAY[0..1] OF LREAL := [2(1000.0000000000)]; (*p2s values for map in [mbar]*)
  END_VAR
  VAR_INPUT
        MapIoP2sy : ARRAY[0..1] OF LREAL := [2(1.0000000000)]; (*integral gain values for map in [CADbfTDC / s / CADafTDC]*)
  END_VAR
  VAR_INPUT
        MapMFB50oT3HPx : ARRAY[0..1] OF LREAL := [2(20.0000000000)]; (*T3HP values for map in [°C]*)
  END_VAR
  VAR_INPUT
        MapMFB50oT3HPy : ARRAY[0..1] OF LREAL := [2(4.0000000000)]; (*MFB50 offset values for map in [CADafTDC]*)
  END_VAR
  VAR_INPUT
        MapMFB50oP2sx : ARRAY[0..1] OF LREAL := [2(1000.0000000000)]; (*p2s values for map in [mbar]*)
  END_VAR
  VAR_INPUT
        MapMFB50oP2sy : ARRAY[0..1] OF LREAL := [2(4.0000000000)]; (*MFB50 offset values for map in [CADafTDC]*)
  END_VAR
  VAR_INPUT
        freezeAllCyl : ARRAY[0..20] OF BOOL := [21(FALSE)]; (*freeze all PI controller outputs and integrators [boolean]*)
  END_VAR
  VAR_INPUT
        uMax : LREAL := 5.0000000000; (*Max limit for IT offset in (CADbfTDC)*)
  END_VAR
  VAR_INPUT
        resetAllCyl : ARRAY[0..20] OF BOOL := [21(FALSE)]; (*reset PI controller of cylinder if = true [boolean]*)
  END_VAR
  VAR_INPUT
        I0AllCyl : ARRAY[0..20] OF LREAL; (*if reset = 1 PI controller of cylinder will be reset to this value [CADbfTDC]*)
  END_VAR
  VAR_INPUT
        MFB50RefOffsetAllCyl : ARRAY[0..20] OF LREAL; (*External offset on reference MFB50 for each cylinder in [CADafTDC]*)
  END_VAR
  VAR_INPUT
        isSkipAllCyl : ARRAY[0..20] OF BOOL := [21(FALSE)]; (*indicator if cylinder is skipped [boolean]*)
  END_VAR
  VAR_INPUT
        isKnockITRetAllCyl : ARRAY[0..20] OF BOOL := [21(FALSE)]; (*indicator if ignition timing on cylinder is retarded due to knock [boolean]*)
  END_VAR
  VAR_INPUT
        isSensFailAllCyl : ARRAY[0..20] OF BOOL := [21(FALSE)]; (*indicator if sensor failure was detected on cylinder [boolean]*)
  END_VAR
  VAR_INPUT
        isITRetLimpHomeAllCyl : ARRAY[0..20] OF BOOL := [21(FALSE)]; (*indicator if ignition timing on cylinder is retarded due to knock [boolean]*)
  END_VAR
  VAR_INPUT
        isFastStart : BOOL := FALSE; (*indicator if fast start is possible [boolean]*)
  END_VAR
  VAR_INPUT
        EngOpState : INT; (*Engine operation state [integer], states 1-5*)
  END_VAR
  VAR_INPUT
        p2s_A : LREAL; (*boost pressure reading bank A in [mbar] *)
  END_VAR
  VAR_INPUT
        uMin : LREAL := -5.0000000000; (*Min limit for IT offset in (CADbfTDC)*)
  END_VAR
  VAR_INPUT
        p2s_B : LREAL; (*boost pressure reading bank B in [mbar]*)
  END_VAR
  VAR_INPUT
        T3HP_A : LREAL; (*Temperature measurement between HP and LP turbines bank A in [°C]*)
  END_VAR
  VAR_INPUT
        T3HP_B : LREAL; (*Temperature measurement between HP and LP turbines bank B in [°C]*)
  END_VAR
  VAR_INPUT
        isLVRT : BOOL := FALSE; (*Indicates LVRT event, impulse for a certain time*)
  END_VAR
  VAR_INPUT
        engSpeed : LREAL := 1000.0000000000; (*engine speed in [rpm]*)
  END_VAR
  VAR_INPUT
        MFB50ActAllCyl : ARRAY[0..20] OF LREAL; (*MFB50 actual value for each cylinder in [CADaFTDC]*)
  END_VAR
  VAR_INPUT
        MFB50EnPowTh : LREAL := 25.0000000000; (*Load threshold for MFB50 control release in [% of  nom load]*)
  END_VAR
  VAR_INPUT
        PelAct : LREAL; (*Actual filtered electric load [% of  nom load]*)
  END_VAR
  VAR_INPUT
        LoadEnabled : BOOL := FALSE; (*If 1, MFB50 control is enabled above load threshold*)
  END_VAR
  VAR_INPUT
        deadbandPos : LREAL; (*Deadband for positive values (CADafTDC)*)
  END_VAR
  VAR_INPUT
        deadbandNeg : LREAL; (*Deadband for negative values (CADafTDC)*)
  END_VAR
  VAR_INPUT
        T1_PT1 : LREAL := 1.0000000000; (*First order time constant for PT1 filter in [s]*)
  END_VAR
  VAR_INPUT
        init_PT1 : ARRAY[0..20] OF LREAL; (*Initial values for PT1 filter for each cylinder in [CADafTDC]*)
  END_VAR
  VAR_INPUT
        MFB50ContrEn : BOOL := TRUE; (*activate MFB50 control if = 1 [boolean], if 0, main control code will not be executed (case loop)*)
  END_VAR
  VAR_INPUT
        MFB50EnSpdTh : LREAL := 500.0000000000; (*speed threshold for MFB50 control release in [rpm]*)
  END_VAR
  VAR_OUTPUT
        MFB50RefGlobP2s : LREAL; (*Reference offset for MFB50 depend on P2s [CADafTDC]*)
  END_VAR
  VAR_OUTPUT
        T3HPout : LREAL := 40.0000000000; (*T3HP value input to MFB50 offset map in [mbar]*)
  END_VAR
  VAR_OUTPUT
        MFB50RefGlobT3HP : LREAL; (*Reference offset for MFB50 depend on T3HP [CADafTDC]*)
  END_VAR
  VAR_OUTPUT
        p2sOut : LREAL := 1000.0000000000; (*p2s value input to MFB50 offset map in [mbar]*)
  END_VAR
  VAR_OUTPUT
        P : LREAL; (*Proportional gain of MFB50 controller*)
  END_VAR
  VAR_OUTPUT
        I : LREAL; (*Integral gain of MFB50 controller*)
  END_VAR
  VAR_OUTPUT
        freezeCyl : BOOL := FALSE; (*cylinder freeze of current calculation ( cyl 1-20)*)
  END_VAR
  VAR_OUTPUT
        cyl : DINT := 1; (*cylinder of current calculation [1-20]*)
  END_VAR
  VAR_OUTPUT
        ITOffsetAllCyl_u : ARRAY[0..20] OF LREAL; (*MFB50 controller output u: IT-offset in [CADbfTDC]*)
  END_VAR
  VAR_OUTPUT
        ITOffsetAllCyl_up : ARRAY[0..20] OF LREAL; (*MFB50 controller proportional output up: IT-offset in [CADbfTDC]*)
  END_VAR
  VAR_OUTPUT
        ITOffsetAllCyl_ui : ARRAY[0..20] OF LREAL; (*MFB50 controller integral output ui: IT-offset in [CADbfTDC]*)
  END_VAR
  VAR_OUTPUT
        clock : DINT; (*MFB50 controller output u: IT-offset in [CADbfTDC]*)
  END_VAR
  VAR_OUTPUT
        MFB50RefGlob : LREAL; (*Global reference for MFB50 in [CADafTDC]*)
  END_VAR
  VAR_OUTPUT
        MFB50ActFiltAllCyl : ARRAY[0..20] OF LREAL; (*Filtered MFB50 actual value in [CADafTDC]*)
  END_VAR
  VAR_OUTPUT
        MFB50MedianFilt : LREAL; (*Filtered Median of MFB50 in [CADafTDC]*)
  END_VAR
  VAR_OUTPUT
        MFB50Median : LREAL; (*Median of MFB50 in [CADafTDC]*)
  END_VAR
  VAR_OUTPUT
        Tcycle : LREAL := 0.1200000000; (*Combustion cycle time in [s]*)
  END_VAR
  VAR_OUTPUT
        ACversion : LREAL := 1.0000000000; (*Autocode version (manually set in Simulink)*)
  END_VAR
	VAR
		bur_BlockIO_MFB50Contr_Lib : BlockIO_MFB50Contr_Lib;
	END_VAR
	VAR
		bur_D_Work_MFB50Contr_Lib : D_Work_MFB50Contr_Lib;
	END_VAR
END_FUNCTION_BLOCK
```

#### lMFB50Cont.typ
```iecst
TYPE

END_TYPE
TYPE
BlockIO_MFB50Contr_Lib : STRUCT
	Divide : LREAL;
	LookupTableDynamic1 : LREAL;
	LookupTableDynamic2 : LREAL;
	p2sOut : LREAL;
	LookupTableDynamic1_m : LREAL;
	LookupTableDynamic : LREAL;
	Add1 : LREAL;
	T3HPout : LREAL;
	out : ARRAY[0..20] OF LREAL;
	up : ARRAY[0..20] OF LREAL;
	ui : ARRAY[0..20] OF LREAL;
	y_f : ARRAY[0..20] OF LREAL;
	y_median : LREAL;
	y_f_e : LREAL;
	DataTypeConversion : DINT;
	DataTypeConversion_o : DINT;
	LogicalOperator : BOOL;
END_STRUCT;
D_Work_MFB50Contr_Lib : STRUCT
	UnitDelay_DSTATE : LREAL;
	iState : ARRAY[0..20] OF LREAL;
	uState : ARRAY[0..20] OF LREAL;
	pState : ARRAY[0..20] OF LREAL;
	y_z : ARRAY[0..20] OF LREAL;
	y_f_z : ARRAY[0..20] OF LREAL;
	y_f_int : ARRAY[0..20] OF LREAL;
	y_z_l : LREAL;
	y_f_z_i : LREAL;
	Relay_Mode : BOOL;
	iState_not_empty : BOOL;
	uState_not_empty : BOOL;
	y_z_not_empty : BOOL;
	y_f_int_not_empty : BOOL;
	y_z_not_empty_p : BOOL;
END_STRUCT;
END_TYPE
```

#### MFB50Contr_Lib.h
```c
/********************************************************************
 * COPYRIGHT -- Bernecker + Rainer Industrie-Elektronik Ges.m.b.H.
 ********************************************************************
 * Program: MFB50Contr_Lib
 * File: MFB50Contr_Lib.h
 * Author: 106001702
 * Created: Wed Nov 09 12:46:00 2011
 ********************************************************************
 * Header for program MFB50Contr_Lib
 ********************************************************************
 * Generated with B&R Automation Studio Target for Simulink V4.2
 * (ERT based)
 ********************************************************************/

#ifndef RTW_HEADER_MFB50Contr_Lib_h_
#define RTW_HEADER_MFB50Contr_Lib_h_
#ifndef MFB50Contr_Lib_COMMON_INCLUDES_
# define MFB50Contr_Lib_COMMON_INCLUDES_
#include <math.h>
#include "rtwtypes.h"
#endif                                 /* MFB50Contr_Lib_COMMON_INCLUDES_ */

#include "MFB50Contr_Lib_types.h"
#include "lMFB50Cont.h"

/* Macros for accessing real-time model data structure */
#ifndef rtmGetErrorStatus
# define rtmGetErrorStatus(rtm)        ((void*) 0)
#endif

#ifndef rtmSetErrorStatus
# define rtmSetErrorStatus(rtm, val)   ((void) 0)
#endif

#ifndef rtmGetStopRequested
# define rtmGetStopRequested(rtm)      ((void*) 0)
#endif

#ifndef MIN
#define MIN(a,b)                       ((a) < (b) ? (a) : (b))
#endif

#ifndef MAX
#define MAX(a,b)                       ((a) > (b) ? (a) : (b))
#endif

/* Block signals (auto storage) */

/* Block states (auto storage) for system '<Root>' */

/* Block signals (auto storage) */
extern BlockIO_MFB50Contr_Lib MFB50Contr_Lib_B;

/* Block states (auto storage) */
extern D_Work_MFB50Contr_Lib MFB50Contr_Lib_DWork;

/* Model entry point functions */
extern void MFB50Contr_Lib_initialize(struct MFB50Contr* inst);
extern void MFB50Contr_Lib_step(struct MFB50Contr* inst);
extern void MFB50Contr_Lib_terminate(struct MFB50Contr* inst);

/*-
 * The generated code includes comments that allow you to trace directly
 * back to the appropriate location in the model.  The basic format
 * is <system>/block_name, where system is the system number (uniquely
 * assigned by Simulink) and block_name is the name of the block.
 *
 * Use the MATLAB hilite_system command to trace the generated code back
 * to the model.  For example,
 *
 * hilite_system('<S3>')    - opens system 3
 * hilite_system('<S3>/Kp') - opens and selects block Kp which resides in S3
 *
 * Here is the system hierarchy for this model
 *
 * '<Root>' : 'MFB50Contr_Lib'
 * '<S1>'   : 'MFB50Contr_Lib/1st order Filter2'
 * '<S2>'   : 'MFB50Contr_Lib/Compare To Zero'
 * '<S3>'   : 'MFB50Contr_Lib/MFB50Controller'
 * '<S4>'   : 'MFB50Contr_Lib/MFB50RefCalc'
 * '<S5>'   : 'MFB50Contr_Lib/Median'
 * '<S6>'   : 'MFB50Contr_Lib/Model Info'
 * '<S7>'   : 'MFB50Contr_Lib/PI cntr gain scheduling'
 * '<S8>'   : 'MFB50Contr_Lib/clockGenerator'
 * '<S9>'   : 'MFB50Contr_Lib/param filter p2'
 * '<S10>'  : 'MFB50Contr_Lib/MFB50Controller/MFB50ContrAllCyl'
 * '<S11>'  : 'MFB50Contr_Lib/MFB50Controller/MFB50ContrAllCyl/1st order Filter'
 * '<S12>'  : 'MFB50Contr_Lib/MFB50Controller/MFB50ContrAllCyl/PI controller'
 * '<S13>'  : 'MFB50Contr_Lib/MFB50Controller/MFB50ContrAllCyl/PI controller/PICntr'
 * '<S14>'  : 'MFB50Contr_Lib/MFB50RefCalc/LVRT control'
 * '<S15>'  : 'MFB50Contr_Lib/MFB50RefCalc/T3HPcalc'
 * '<S16>'  : 'MFB50Contr_Lib/PI cntr gain scheduling/P2sCalc'
 */
#endif                                 /* RTW_HEADER_MFB50Contr_Lib_h_ */
```
